SPLINE
SPL {X  -165.650, Y  +561.960, Z    +0.000, E1   +45.285, E3 +336665.881}
SPL {X  -165.650, Y  +554.065, Z    +0.000, E1   +45.254, E3 +336681.943}
SPL {X  -165.650, Y  +548.074, Z    +0.000, E1   +45.245, E3 +336694.053}
SPL {X  -165.650, Y  +542.958, Z    +0.000, E1   +45.131, E3 +336705.184}
SPL {X  -165.650, Y  +535.288, Z    +0.000, E1   +45.332, E3 +336719.625}
SPL {X  -165.650, Y  +529.160, Z    +0.000, E1   +45.215, E3 +336732.606}
SPL {X  -165.650, Y  +522.672, Z    +0.000, E1   +45.331, E3 +336745.172}
SPL {X  -165.650, Y  +516.211, Z    +0.000, E1   +45.175, E3 +336759.131}
SPL {X  -165.650, Y  +509.762, Z    +0.000, E1   +45.191, E3 +336772.174}
SPL {X  -165.650, Y  +503.812, Z    +0.000, E1   +45.188, E3 +336784.212}
SPL {X  -165.650, Y  +499.646, Z    +0.000, E1   +44.886, E3 +336794.483}
ENDSPLINE

SPLINE
SPL {X  -165.650, Y  +516.930, Z    +0.000, E1   +36.544, E3 +336803.154}
ENDSPLINE

SPLINE
SPL {X  -165.650, Y  +511.324, Z    +0.000, E1   +37.254, E3 +336814.145}
SPL {X  -165.650, Y  +504.742, Z    +0.000, E1   +38.087, E3 +336826.450}
SPL {X  -165.650, Y  +497.845, Z    +0.000, E1   +39.022, E3 +336838.525}
SPL {X  -165.650, Y  +488.971, Z    +0.000, E1   +40.149, E3 +336853.745}
SPL {X  -165.650, Y  +478.382, Z    +0.000, E1   +41.628, E3 +336869.943}
SPL {X  -165.650, Y  +472.112, Z    +0.000, E1   +42.202, E3 +336880.682}
SPL {X  -165.650, Y  +466.741, Z    +0.000, E1   +42.890, E3 +336888.603}
SPL {X  -165.650, Y  +458.202, Z    +0.000, E1   +44.020, E3 +336900.390}
SPL {X  -165.650, Y  +449.099, Z    +0.000, E1   +44.871, E3 +336914.353}
SPL {X  -165.650, Y  +442.120, Z    +0.000, E1   +45.313, E3 +336925.905}
SPL {X  -165.650, Y  +436.063, Z    +0.000, E1   +44.972, E3 +336940.489}
SPL {X  -165.650, Y  +427.943, Z    +0.000, E1   +45.362, E3 +336954.526}
SPL {X  -165.650, Y  +422.523, Z    +0.000, E1   +45.103, E3 +336967.205}
SPL {X  -165.650, Y  +415.564, Z    +0.000, E1   +45.195, E3 +336980.744}
SPL {X  -165.650, Y  +410.687, Z    +0.000, E1   +44.955, E3 +336992.060}
SPL {X  -165.650, Y  +405.522, Z    +0.000, E1   +45.119, E3 +337001.620}
SPL {X  -165.650, Y  +399.216, Z    +0.000, E1   +45.246, E3 +337013.814}
SPL {X  -165.650, Y  +391.618, Z    +0.000, E1   +45.037, E3 +337030.592}
SPL {X  -165.650, Y  +383.700, Z    +0.000, E1   +45.345, E3 +337044.718}
SPL {X  -165.650, Y  +379.225, Z    +0.000, E1   +45.073, E3 +337055.407}
SPL {X  -165.591, Y  +374.097, Z    +0.000, E1   +45.069, E3 +337065.888}
SPL {X  -165.372, Y  +368.914, Z    +0.000, E1   +45.103, E3 +337076.248}
SPL {X  -164.987, Y  +363.696, Z    +0.000, E1   +45.006, E3 +337087.471}
SPL {X  -164.256, Y  +357.053, Z    +0.000, E1   +44.969, E3 +337101.274}
SPL {X  -163.441, Y  +351.538, Z    +0.000, E1   +44.749, E3 +337113.638}
SPL {X  -162.419, Y  +345.942, Z    +0.000, E1   +44.540, E3 +337126.369}
SPL {X  -161.210, Y  +340.404, Z    +0.000, E1   +44.250, E3 +337139.194}
SPL {X  -159.961, Y  +335.460, Z    +0.000, E1   +44.205, E3 +337149.557}
SPL {X  -158.595, Y  +330.672, Z    +0.000, E1   +43.797, E3 +337161.535}
SPL {X  -157.207, Y  +326.289, Z    +0.000, E1   +43.631, E3 +337171.288}
SPL {X  -152.192, Y  +313.097, Z    +0.000, E1   +47.715, E3 +337174.842}
SPL {X  -146.385, Y  +300.967, Z    +0.000, E1   +50.402, E3 +337181.037}
SPL {X  -138.435, Y  +287.529, Z    +0.000, E1   +45.834, E3 +337242.993}
SPL {X  -134.645, Y  +282.008, Z    +0.000, E1   +45.207, E3 +337272.650}
ENDSPLINE

SPLINE
SPL {X  -154.915, Y  +319.839, Z    +0.000, E1   +31.584, E3 +337332.169}
SPL {X  -161.387, Y  +341.161, Z    +0.000, E1   +22.590, E3 +337346.014}
SPL {X  -164.566, Y  +359.576, Z    +0.000, E1   +13.425, E3 +337324.608}
SPL {X  -165.355, Y  +368.611, Z    +0.000, E1    +8.407, E3 +337328.189}
SPL {X  -165.614, Y  +375.050, Z    +0.000, E1    +4.520, E3 +337329.492}
SPL {X  -165.650, Y  +379.847, Z    +0.000, E1    +1.364, E3 +337327.842}
SPL {X  -165.650, Y  +383.246, Z    +0.000, E1    -1.216, E3 +337326.935}
SPL {X  -165.650, Y  +386.866, Z    +0.000, E1    -4.337, E3 +337326.988}
SPL {X  -165.650, Y  +394.200, Z    +0.000, E1   -11.943, E3 +337324.755}
SPL {X  -165.650, Y  +405.401, Z    +0.000, E1   -24.512, E3 +337324.575}
SPL {X  -165.650, Y  +418.038, Z    +0.000, E1   -38.688, E3 +337320.802}
SPL {X  -165.650, Y  +461.620, Z    +0.000, E1   -55.594, E3 +337340.981}
SPL {X  -165.650, Y  +498.574, Z    +0.000, E1   -52.082, E3 +337402.006}
ENDSPLINE

SPLINE
SPL {X  -165.650, Y  +484.983, Z    +0.000, E1   -45.406, E3 +337417.509}
ENDSPLINE

SPLINE
SPL {X  -165.650, Y  +492.090, Z    +0.000, E1   -45.292, E3 +337432.532}
SPL {X  -165.650, Y  +498.857, Z    +0.000, E1   -45.339, E3 +337445.869}
SPL {X  -165.650, Y  +505.115, Z    +0.000, E1   -45.299, E3 +337458.817}
SPL {X  -165.650, Y  +510.931, Z    +0.000, E1   -45.250, E3 +337470.808}
SPL {X  -165.650, Y  +516.157, Z    +0.000, E1   -45.240, E3 +337481.482}
SPL {X  -165.650, Y  +521.049, Z    +0.000, E1   -45.236, E3 +337491.435}
SPL {X  -165.650, Y  +527.050, Z    +0.000, E1   -45.345, E3 +337502.931}
SPL {X  -165.650, Y  +532.042, Z    +0.000, E1   -45.233, E3 +337513.674}
SPL {X  -165.650, Y  +537.290, Z    +0.000, E1   -45.204, E3 +337524.515}
SPL {X  -165.650, Y  +544.196, Z    +0.000, E1   -45.432, E3 +337537.189}
SPL {X  -165.650, Y  +548.678, Z    +0.000, E1   -45.162, E3 +337547.753}
SPL {X  -165.650, Y  +554.600, Z    +0.000, E1   -45.345, E3 +337558.730}
SPL {X  -165.650, Y  +559.896, Z    +0.000, E1   -45.150, E3 +337570.585}
SPL {X  -165.650, Y  +566.830, Z    +0.000, E1   -45.346, E3 +337583.566}
SPL {X  -165.650, Y  +573.074, Z    +0.000, E1   -45.379, E3 +337595.896}
SPL {X  -165.650, Y  +579.360, Z    +0.000, E1   -45.300, E3 +337609.181}
SPL {X  -165.650, Y  +584.577, Z    +0.000, E1   -45.167, E3 +337620.405}
SPL {X  -165.650, Y  +590.060, Z    +0.000, E1   -45.221, E3 +337631.295}
SPL {X  -165.650, Y  +596.611, Z    +0.000, E1   -45.390, E3 +337643.532}
SPL {X  -165.650, Y  +601.960, Z    +0.000, E1   -45.255, E3 +337655.140}
SPL {X  -165.650, Y  +605.976, Z    +0.000, E1   -45.260, E3 +337663.190}
SPL {X  -165.650, Y  +610.850, Z    +0.000, E1   -45.208, E3 +337673.459}
SPL {X  -165.650, Y  +617.450, Z    +0.000, E1   -45.402, E3 +337685.661}
SPL {X  -165.650, Y  +622.720, Z    +0.000, E1   -45.272, E3 +337697.059}
SPL {X  -165.650, Y  +627.828, Z    +0.000, E1   -45.174, E3 +337708.015}
SPL {X  -165.650, Y  +634.620, Z    +0.000, E1   -45.438, E3 +337720.221}
SPL {X  -165.650, Y  +640.808, Z    +0.000, E1   -45.294, E3 +337733.596}
SPL {X  -165.650, Y  +646.552, Z    +0.000, E1   -45.137, E3 +337746.120}
SPL {X  -165.650, Y  +652.431, Z    +0.000, E1   -45.333, E3 +337756.874}
SPL {X  -165.650, Y  +657.443, Z    +0.000, E1   -45.316, E3 +337767.131}
SPL {X  -165.650, Y  +662.999, Z    +0.000, E1   -45.214, E3 +337779.003}
SPL {X  -165.650, Y  +668.737, Z    +0.000, E1   -45.236, E3 +337790.518}
SPL {X  -165.650, Y  +675.226, Z    +0.000, E1   -45.503, E3 +337802.021}
SPL {X  -165.597, Y  +679.672, Z    +0.000, E1   -45.206, E3 +337812.742}
SPL {X  -165.388, Y  +684.808, Z    +0.000, E1   -45.192, E3 +337823.250}
SPL {X  -165.020, Y  +689.938, Z    +0.000, E1   -45.107, E3 +337834.193}
SPL {X  -164.358, Y  +696.147, Z    +0.000, E1   -45.160, E3 +337846.458}
SPL {X  -163.631, Y  +701.286, Z    +0.000, E1   -44.994, E3 +337857.751}
SPL {X  -163.047, Y  +704.748, Z    +0.000, E1   -44.682, E3 +337866.574}
SPL {X  -161.884, Y  +710.619, Z    +0.000, E1   -44.738, E3 +337878.199}
SPL {X  -160.692, Y  +715.726, Z    +0.000, E1   -44.379, E3 +337890.522}
SPL {X  -159.384, Y  +720.631, Z    +0.000, E1   -44.155, E3 +337901.672}
SPL {X  -157.745, Y  +726.062, Z    +0.000, E1   -43.902, E3 +337914.158}
SPL {X  -153.030, Y  +738.918, Z    +0.000, E1   -47.123, E3 +337921.761}
SPL {X  -145.149, Y  +755.323, Z    +0.000, E1   -51.167, E3 +337927.893}
SPL {X  -144.116, Y  +757.172, Z    +0.000, E1   -42.809, E3 +337994.443}
SPL {X  -127.227, Y  +781.582, Z    +0.000, E1   -46.780, E3 +338040.112}
ENDSPLINE

SPLINE
SPL {X  -133.736, Y  +773.248, Z    +0.000, E1   -45.385, E3 +338118.155}
SPL {X  -160.761, Y  +715.447, Z    +0.000, E1   -23.748, E3 +338075.004}
SPL {X  -164.304, Y  +696.571, Z    +0.000, E1   -14.525, E3 +338080.228}
SPL {X  -165.498, Y  +682.585, Z    +0.000, E1    -6.769, E3 +338079.903}
SPL {X  -165.650, Y  +674.975, Z    +0.000, E1    -1.888, E3 +338078.261}
SPL {X  -165.650, Y  +670.481, Z    +0.000, E1    +1.454, E3 +338077.702}
SPL {X  -165.650, Y  +665.304, Z    +0.000, E1    +6.303, E3 +338076.205}
SPL {X  -165.650, Y  +657.587, Z    +0.000, E1   +14.733, E3 +338074.979}
SPL {X  -165.650, Y  +646.511, Z    +0.000, E1   +26.434, E3 +338077.540}
SPL {X  -165.650, Y  +637.905, Z    +0.000, E1   +40.225, E3 +338065.665}
SPL {X  -165.650, Y  +607.385, Z    +0.000, E1   +51.775, E3 +338085.423}
SPL {X  -165.650, Y  +598.058, Z    +0.000, E1   +51.157, E3 +338098.884}
SPL {X  -165.650, Y  +553.219, Z    +0.000, E1   +52.865, E3 +338153.067}
ENDSPLINE

SPLINE
SPL {X  -165.650, Y  +569.883, Z    +0.000, E1   +45.183, E3 +338168.744}
ENDSPLINE

SPLINE
SPL {X  -165.650, Y  +564.081, Z    +0.000, E1   +45.208, E3 +338180.361}
SPL {X  -165.650, Y  +557.350, Z    +0.000, E1   +45.265, E3 +338193.798}
SPL {X  -165.650, Y  +549.414, Z    +0.000, E1   +45.294, E3 +338209.700}
SPL {X  -165.650, Y  +542.958, Z    +0.000, E1   +45.131, E3 +338223.702}
SPL {X  -165.650, Y  +535.288, Z    +0.000, E1   +45.332, E3 +338238.143}
SPL {X  -165.650, Y  +528.026, Z    +0.000, E1   +45.173, E3 +338253.802}
SPL {X  -165.650, Y  +519.896, Z    +0.000, E1   +45.366, E3 +338269.141}
SPL {X  -165.650, Y  +512.740, Z    +0.000, E1   +45.225, E3 +338284.488}
SPL {X  -165.650, Y  +505.100, Z    +0.000, E1   +45.197, E3 +338300.171}
SPL {X  -165.650, Y  +499.646, Z    +0.000, E1   +44.886, E3 +338313.002}
ENDSPLINE

SPLINE
SPL {X  -165.650, Y  +516.930, Z    +0.000, E1   +36.544, E3 +338321.672}
ENDSPLINE

SPLINE
SPL {X  -165.650, Y  +511.324, Z    +0.000, E1   +37.254, E3 +338332.663}
SPL {X  -165.650, Y  +502.734, Z    +0.000, E1   +38.389, E3 +338348.432}
SPL {X  -165.650, Y  +493.826, Z    +0.000, E1   +39.521, E3 +338364.094}
SPL {X  -165.650, Y  +485.086, Z    +0.000, E1   +40.678, E3 +338378.407}
SPL {X  -165.650, Y  +474.980, Z    +0.000, E1   +42.004, E3 +338394.034}
SPL {X  -165.650, Y  +463.933, Z    +0.000, E1   +43.299, E3 +338410.920}
SPL {X  -165.650, Y  +452.327, Z    +0.000, E1   +44.758, E3 +338426.826}
SPL {X  -165.650, Y  +444.380, Z    +0.000, E1   +45.056, E3 +338441.421}
SPL {X  -165.650, Y  +436.063, Z    +0.000, E1   +44.972, E3 +338459.008}
SPL {X  -165.650, Y  +427.943, Z    +0.000, E1   +45.362, E3 +338473.045}
SPL {X  -165.650, Y  +422.523, Z    +0.000, E1   +45.103, E3 +338485.723}
SPL {X  -165.650, Y  +415.564, Z    +0.000, E1   +45.195, E3 +338499.262}
SPL {X  -165.650, Y  +410.687, Z    +0.000, E1   +44.955, E3 +338510.578}
SPL {X  -165.650, Y  +405.522, Z    +0.000, E1   +45.119, E3 +338520.138}
SPL {X  -165.650, Y  +399.216, Z    +0.000, E1   +45.246, E3 +338532.332}
SPL {X  -165.650, Y  +391.618, Z    +0.000, E1   +45.037, E3 +338549.110}
SPL {X  -165.650, Y  +383.700, Z    +0.000, E1   +45.345, E3 +338563.237}
SPL {X  -165.650, Y  +379.225, Z    +0.000, E1   +45.073, E3 +338573.926}
SPL {X  -165.591, Y  +374.097, Z    +0.000, E1   +45.069, E3 +338584.407}
SPL {X  -165.372, Y  +368.914, Z    +0.000, E1   +45.103, E3 +338594.767}
SPL {X  -164.833, Y  +362.064, Z    +0.000, E1   +44.999, E3 +338609.552}
SPL {X  -164.024, Y  +355.348, Z    +0.000, E1   +45.002, E3 +338622.940}
SPL {X  -163.140, Y  +349.774, Z    +0.000, E1   +44.687, E3 +338636.327}
SPL {X  -162.065, Y  +344.224, Z    +0.000, E1   +44.509, E3 +338648.417}
SPL {X  -161.210, Y  +340.404, Z    +0.000, E1   +44.250, E3 +338657.713}
SPL {X  -159.961, Y  +335.460, Z    +0.000, E1   +44.205, E3 +338668.076}
SPL {X  -158.595, Y  +330.672, Z    +0.000, E1   +43.797, E3 +338680.054}
SPL {X  -157.207, Y  +326.289, Z    +0.000, E1   +43.631, E3 +338689.807}
SPL {X  -152.192, Y  +313.097, Z    +0.000, E1   +47.715, E3 +338693.361}
SPL {X  -146.385, Y  +300.967, Z    +0.000, E1   +50.402, E3 +338699.556}
SPL {X  -138.435, Y  +287.529, Z    +0.000, E1   +45.834, E3 +338761.512}
SPL {X  -134.645, Y  +282.008, Z    +0.000, E1   +45.207, E3 +338791.168}
ENDSPLINE

SPLINE
SPL {X  -154.915, Y  +319.839, Z    +0.000, E1   +31.584, E3 +338850.687}
SPL {X  -161.387, Y  +341.161, Z    +0.000, E1   +22.590, E3 +338864.533}
SPL {X  -164.566, Y  +359.576, Z    +0.000, E1   +13.425, E3 +338843.126}
SPL {X  -165.355, Y  +368.611, Z    +0.000, E1    +8.407, E3 +338846.707}
SPL {X  -165.614, Y  +375.050, Z    +0.000, E1    +4.520, E3 +338848.011}
SPL {X  -165.650, Y  +379.271, Z    +0.000, E1    +1.752, E3 +338845.032}
SPL {X  -165.650, Y  +382.603, Z    +0.000, E1    -0.657, E3 +338846.240}
SPL {X  -165.650, Y  +386.866, Z    +0.000, E1    -4.337, E3 +338845.506}
SPL {X  -165.650, Y  +392.464, Z    +0.000, E1   -10.170, E3 +338843.510}
SPL {X  -165.650, Y  +397.361, Z    +0.000, E1   -15.736, E3 +338842.842}
SPL {X  -165.650, Y  +404.553, Z    +0.000, E1   -23.488, E3 +338843.618}
SPL {X  -165.650, Y  +415.773, Z    +0.000, E1   -36.308, E3 +338839.770}
SPL {X  -165.650, Y  +461.620, Z    +0.000, E1   -55.594, E3 +338859.499}
SPL {X  -165.650, Y  +505.847, Z    +0.000, E1   -55.467, E3 +338911.472}
ENDSPLINE

SPLINE
SPL {X  -165.650, Y  +495.538, Z    +0.000, E1   -50.621, E3 +338923.956}
SPL {X  -165.650, Y  +483.168, Z    +0.000, E1   -45.573, E3 +338931.182}
ENDSPLINE

SPLINE
SPL {X  -165.650, Y  +487.615, Z    +0.000, E1   -45.254, E3 +338942.203}
SPL {X  -165.650, Y  +493.602, Z    +0.000, E1   -45.283, E3 +338954.043}
SPL {X  -165.650, Y  +498.857, Z    +0.000, E1   -45.339, E3 +338964.387}
SPL {X  -165.650, Y  +504.159, Z    +0.000, E1   -45.384, E3 +338974.782}
SPL {X  -165.650, Y  +509.628, Z    +0.000, E1   -45.217, E3 +338986.965}
SPL {X  -165.650, Y  +516.157, Z    +0.000, E1   -45.240, E3 +339000.000}
SPL {X  -165.650, Y  +521.049, Z    +0.000, E1   -45.236, E3 +339009.953}
SPL {X  -165.650, Y  +527.050, Z    +0.000, E1   -45.345, E3 +339021.449}
SPL {X  -165.650, Y  +532.042, Z    +0.000, E1   -45.233, E3 +339032.193}
SPL {X  -165.650, Y  +537.290, Z    +0.000, E1   -45.204, E3 +339043.033}
SPL {X  -165.650, Y  +544.196, Z    +0.000, E1   -45.432, E3 +339055.708}
SPL {X  -165.650, Y  +548.678, Z    +0.000, E1   -45.162, E3 +339066.271}
SPL {X  -165.650, Y  +554.600, Z    +0.000, E1   -45.345, E3 +339077.249}
SPL {X  -165.650, Y  +559.896, Z    +0.000, E1   -45.150, E3 +339089.104}
SPL {X  -165.650, Y  +566.830, Z    +0.000, E1   -45.346, E3 +339102.084}
SPL {X  -165.650, Y  +573.074, Z    +0.000, E1   -45.379, E3 +339114.415}
SPL {X  -165.650, Y  +577.292, Z    +0.000, E1   -45.246, E3 +339123.678}
SPL {X  -165.650, Y  +583.131, Z    +0.000, E1   -45.255, E3 +339135.620}
SPL {X  -165.650, Y  +590.060, Z    +0.000, E1   -45.221, E3 +339149.814}
SPL {X  -165.650, Y  +596.611, Z    +0.000, E1   -45.390, E3 +339162.050}
SPL {X  -165.650, Y  +603.637, Z    +0.000, E1   -45.296, E3 +339176.969}
SPL {X  -165.650, Y  +610.850, Z    +0.000, E1   -45.208, E3 +339191.977}
SPL {X  -165.650, Y  +617.450, Z    +0.000, E1   -45.402, E3 +339204.180}
SPL {X  -165.650, Y  +622.720, Z    +0.000, E1   -45.272, E3 +339215.577}
SPL {X  -165.650, Y  +627.828, Z    +0.000, E1   -45.174, E3 +339226.534}
SPL {X  -165.650, Y  +636.061, Z    +0.000, E1   -45.380, E3 +339242.196}
SPL {X  -165.650, Y  +645.149, Z    +0.000, E1   -45.285, E3 +339261.127}
SPL {X  -165.650, Y  +652.431, Z    +0.000, E1   -45.333, E3 +339275.393}
SPL {X  -165.650, Y  +657.443, Z    +0.000, E1   -45.316, E3 +339285.649}
SPL {X  -165.650, Y  +662.999, Z    +0.000, E1   -45.214, E3 +339297.521}
SPL {X  -165.650, Y  +668.737, Z    +0.000, E1   -45.236, E3 +339309.036}
SPL {X  -165.650, Y  +675.226, Z    +0.000, E1   -45.503, E3 +339320.540}
SPL {X  -165.597, Y  +679.672, Z    +0.000, E1   -45.206, E3 +339331.261}
SPL {X  -165.388, Y  +684.808, Z    +0.000, E1   -45.192, E3 +339341.768}
SPL {X  -165.020, Y  +689.938, Z    +0.000, E1   -45.107, E3 +339352.711}
SPL {X  -164.358, Y  +696.147, Z    +0.000, E1   -45.160, E3 +339364.977}
SPL {X  -163.631, Y  +701.286, Z    +0.000, E1   -44.994, E3 +339376.269}
SPL {X  -163.047, Y  +704.748, Z    +0.000, E1   -44.682, E3 +339385.093}
SPL {X  -161.884, Y  +710.619, Z    +0.000, E1   -44.738, E3 +339396.718}
SPL {X  -160.692, Y  +715.726, Z    +0.000, E1   -44.379, E3 +339409.040}
SPL {X  -158.938, Y  +722.175, Z    +0.000, E1   -44.121, E3 +339423.688}
SPL {X  -156.604, Y  +729.490, Z    +0.000, E1   -44.229, E3 +339437.678}
SPL {X  -147.100, Y  +751.668, Z    +0.000, E1   -50.624, E3 +339443.565}
SPL {X  -143.038, Y  +759.047, Z    +0.000, E1   -43.157, E3 +339515.585}
SPL {X  -123.277, Y  +786.146, Z    +0.000, E1   -47.533, E3 +339571.640}
ENDSPLINE

SPLINE
SPL {X  -133.736, Y  +773.248, Z    +0.000, E1   -45.385, E3 +339636.673}
SPL {X  -160.761, Y  +715.447, Z    +0.000, E1   -23.748, E3 +339593.523}
SPL {X  -164.304, Y  +696.571, Z    +0.000, E1   -14.525, E3 +339598.747}
SPL {X  -165.374, Y  +685.052, Z    +0.000, E1    -8.166, E3 +339598.140}
SPL {X  -165.648, Y  +676.230, Z    +0.000, E1    -2.814, E3 +339597.292}
SPL {X  -165.650, Y  +670.481, Z    +0.000, E1    +1.454, E3 +339596.221}
SPL {X  -165.650, Y  +665.304, Z    +0.000, E1    +6.303, E3 +339594.723}
SPL {X  -165.650, Y  +657.587, Z    +0.000, E1   +14.733, E3 +339593.498}
SPL {X  -165.650, Y  +646.511, Z    +0.000, E1   +26.434, E3 +339596.059}
SPL {X  -165.650, Y  +637.905, Z    +0.000, E1   +40.225, E3 +339584.183}
SPL {X  -165.650, Y  +607.385, Z    +0.000, E1   +51.775, E3 +339603.941}
SPL {X  -165.650, Y  +598.058, Z    +0.000, E1   +51.157, E3 +339617.403}
SPL {X  -165.650, Y  +553.656, Z    +0.000, E1   +53.998, E3 +339664.402}
SPL {X  -165.650, Y  +553.154, Z    +0.000, E1   +52.102, E3 +339675.929}
ENDSPLINE

SPLINE
SPL {X  -165.650, Y  +569.883, Z    +0.000, E1   +45.183, E3 +339687.262}
ENDSPLINE

SPLINE
SPL {X  -165.650, Y  +564.081, Z    +0.000, E1   +45.208, E3 +339698.880}
SPL {X  -165.650, Y  +557.350, Z    +0.000, E1   +45.265, E3 +339712.317}
SPL {X  -165.650, Y  +549.414, Z    +0.000, E1   +45.294, E3 +339728.219}
SPL {X  -165.650, Y  +542.958, Z    +0.000, E1   +45.131, E3 +339742.221}
SPL {X  -165.650, Y  +535.288, Z    +0.000, E1   +45.332, E3 +339756.662}
SPL {X  -165.650, Y  +528.026, Z    +0.000, E1   +45.173, E3 +339772.320}
SPL {X  -165.650, Y  +520.964, Z    +0.000, E1   +45.458, E3 +339784.825}
SPL {X  -165.650, Y  +516.211, Z    +0.000, E1   +45.175, E3 +339796.168}
SPL {X  -165.650, Y  +509.762, Z    +0.000, E1   +45.191, E3 +339809.211}
SPL {X  -165.650, Y  +503.812, Z    +0.000, E1   +45.188, E3 +339821.249}
SPL {X  -165.650, Y  +499.646, Z    +0.000, E1   +44.886, E3 +339831.520}
ENDSPLINE

SPLINE
SPL {X  -165.650, Y  +516.930, Z    +0.000, E1   +36.544, E3 +339840.191}
ENDSPLINE

SPLINE
SPL {X  -165.650, Y  +511.324, Z    +0.000, E1   +37.254, E3 +339851.182}
SPL {X  -165.650, Y  +504.742, Z    +0.000, E1   +38.087, E3 +339863.487}
SPL {X  -165.650, Y  +497.845, Z    +0.000, E1   +39.022, E3 +339875.562}
SPL {X  -165.650, Y  +488.971, Z    +0.000, E1   +40.149, E3 +339890.783}
SPL {X  -165.650, Y  +478.382, Z    +0.000, E1   +41.628, E3 +339906.980}
SPL {X  -165.650, Y  +472.112, Z    +0.000, E1   +42.202, E3 +339917.719}
SPL {X  -165.650, Y  +466.741, Z    +0.000, E1   +42.890, E3 +339925.640}
SPL {X  -165.650, Y  +458.202, Z    +0.000, E1   +44.020, E3 +339937.427}
SPL {X  -165.650, Y  +449.099, Z    +0.000, E1   +44.871, E3 +339951.390}
SPL {X  -165.650, Y  +442.120, Z    +0.000, E1   +45.313, E3 +339962.942}
SPL {X  -165.650, Y  +436.063, Z    +0.000, E1   +44.972, E3 +339977.526}
SPL {X  -165.650, Y  +427.943, Z    +0.000, E1   +45.362, E3 +339991.563}
SPL {X  -165.650, Y  +422.523, Z    +0.000, E1   +45.103, E3 +340004.242}
SPL {X  -165.650, Y  +415.564, Z    +0.000, E1   +45.195, E3 +340017.781}
SPL {X  -165.650, Y  +410.687, Z    +0.000, E1   +44.955, E3 +340029.097}
SPL {X  -165.650, Y  +405.522, Z    +0.000, E1   +45.119, E3 +340038.657}
SPL {X  -165.650, Y  +400.300, Z    +0.000, E1   +45.439, E3 +340047.341}
SPL {X  -165.650, Y  +396.171, Z    +0.000, E1   +44.969, E3 +340058.598}
SPL {X  -165.650, Y  +390.060, Z    +0.000, E1   +45.007, E3 +340070.832}
SPL {X  -165.650, Y  +383.700, Z    +0.000, E1   +45.345, E3 +340081.755}
SPL {X  -165.650, Y  +379.225, Z    +0.000, E1   +45.073, E3 +340092.444}
SPL {X  -165.591, Y  +374.097, Z    +0.000, E1   +45.069, E3 +340102.926}
SPL {X  -165.372, Y  +368.914, Z    +0.000, E1   +45.103, E3 +340113.285}
SPL {X  -164.833, Y  +362.064, Z    +0.000, E1   +44.999, E3 +340128.070}
SPL {X  -164.024, Y  +355.348, Z    +0.000, E1   +45.002, E3 +340141.459}
SPL {X  -163.441, Y  +351.538, Z    +0.000, E1   +44.749, E3 +340150.675}
SPL {X  -162.419, Y  +345.942, Z    +0.000, E1   +44.540, E3 +340163.406}
SPL {X  -161.210, Y  +340.404, Z    +0.000, E1   +44.250, E3 +340176.231}
SPL {X  -159.961, Y  +335.460, Z    +0.000, E1   +44.205, E3 +340186.594}
SPL {X  -158.595, Y  +330.672, Z    +0.000, E1   +43.797, E3 +340198.572}
SPL {X  -156.695, Y  +324.773, Z    +0.000, E1   +43.987, E3 +340209.469}
SPL {X  -148.318, Y  +304.733, Z    +0.000, E1   +49.897, E3 +340214.706}
SPL {X  -137.641, Y  +286.333, Z    +0.000, E1   +45.396, E3 +340289.566}
SPL {X  -137.518, Y  +286.149, Z    +0.000, E1   +42.648, E3 +340362.075}
ENDSPLINE

SPLINE
SPL {X  -156.430, Y  +324.005, Z    +0.000, E1   +29.926, E3 +340367.210}
SPL {X  -161.387, Y  +341.161, Z    +0.000, E1   +22.590, E3 +340383.051}
SPL {X  -164.566, Y  +359.576, Z    +0.000, E1   +13.425, E3 +340361.645}
SPL {X  -165.355, Y  +368.611, Z    +0.000, E1    +8.407, E3 +340365.226}
SPL {X  -165.614, Y  +375.050, Z    +0.000, E1    +4.520, E3 +340366.529}
SPL {X  -165.650, Y  +379.271, Z    +0.000, E1    +1.752, E3 +340363.551}
SPL {X  -165.650, Y  +382.603, Z    +0.000, E1    -0.657, E3 +340364.759}
SPL {X  -165.650, Y  +386.866, Z    +0.000, E1    -4.337, E3 +340364.025}
SPL {X  -165.650, Y  +394.200, Z    +0.000, E1   -11.943, E3 +340361.792}
SPL {X  -165.650, Y  +405.401, Z    +0.000, E1   -24.512, E3 +340361.612}
SPL {X  -165.650, Y  +418.038, Z    +0.000, E1   -38.688, E3 +340357.839}
SPL {X  -165.650, Y  +461.620, Z    +0.000, E1   -55.594, E3 +340378.018}
SPL {X  -165.650, Y  +498.574, Z    +0.000, E1   -52.082, E3 +340439.043}
ENDSPLINE

SPLINE
SPL {X  -165.650, Y  +483.168, Z    +0.000, E1   -45.573, E3 +340449.700}
ENDSPLINE

SPLINE
SPL {X  -165.650, Y  +487.615, Z    +0.000, E1   -45.254, E3 +340460.722}
SPL {X  -165.650, Y  +493.602, Z    +0.000, E1   -45.283, E3 +340472.562}
SPL {X  -165.650, Y  +498.857, Z    +0.000, E1   -45.339, E3 +340482.906}
SPL {X  -165.650, Y  +504.159, Z    +0.000, E1   -45.384, E3 +340493.300}
SPL {X  -165.650, Y  +509.628, Z    +0.000, E1   -45.217, E3 +340505.483}
SPL {X  -165.650, Y  +516.157, Z    +0.000, E1   -45.240, E3 +340518.519}
SPL {X  -165.650, Y  +521.049, Z    +0.000, E1   -45.236, E3 +340528.472}
SPL {X  -165.650, Y  +527.050, Z    +0.000, E1   -45.345, E3 +340539.968}
SPL {X  -165.650, Y  +532.042, Z    +0.000, E1   -45.233, E3 +340550.711}
SPL {X  -165.650, Y  +537.290, Z    +0.000, E1   -45.204, E3 +340561.552}
SPL {X  -165.650, Y  +544.196, Z    +0.000, E1   -45.432, E3 +340574.226}
SPL {X  -165.650, Y  +548.678, Z    +0.000, E1   -45.162, E3 +340584.790}
SPL {X  -165.650, Y  +554.600, Z    +0.000, E1   -45.345, E3 +340595.767}
SPL {X  -165.650, Y  +559.896, Z    +0.000, E1   -45.150, E3 +340607.622}
SPL {X  -165.650, Y  +566.830, Z    +0.000, E1   -45.346, E3 +340620.603}
SPL {X  -165.650, Y  +573.074, Z    +0.000, E1   -45.379, E3 +340632.933}
SPL {X  -165.650, Y  +579.360, Z    +0.000, E1   -45.300, E3 +340646.218}
SPL {X  -165.650, Y  +584.577, Z    +0.000, E1   -45.167, E3 +340657.442}
SPL {X  -165.650, Y  +590.060, Z    +0.000, E1   -45.221, E3 +340668.333}
SPL {X  -165.650, Y  +596.611, Z    +0.000, E1   -45.390, E3 +340680.569}
SPL {X  -165.650, Y  +601.960, Z    +0.000, E1   -45.255, E3 +340692.177}
SPL {X  -165.650, Y  +605.976, Z    +0.000, E1   -45.260, E3 +340700.227}
SPL {X  -165.650, Y  +610.850, Z    +0.000, E1   -45.208, E3 +340710.496}
SPL {X  -165.650, Y  +617.450, Z    +0.000, E1   -45.402, E3 +340722.698}
SPL {X  -165.650, Y  +622.720, Z    +0.000, E1   -45.272, E3 +340734.096}
SPL {X  -165.650, Y  +627.828, Z    +0.000, E1   -45.174, E3 +340745.053}
SPL {X  -165.650, Y  +634.620, Z    +0.000, E1   -45.438, E3 +340757.258}
SPL {X  -165.650, Y  +640.808, Z    +0.000, E1   -45.294, E3 +340770.633}
SPL {X  -165.650, Y  +646.552, Z    +0.000, E1   -45.137, E3 +340783.157}
SPL {X  -165.650, Y  +652.431, Z    +0.000, E1   -45.333, E3 +340793.911}
SPL {X  -165.650, Y  +657.443, Z    +0.000, E1   -45.316, E3 +340804.168}
SPL {X  -165.650, Y  +662.999, Z    +0.000, E1   -45.214, E3 +340816.040}
SPL {X  -165.650, Y  +668.737, Z    +0.000, E1   -45.236, E3 +340827.555}
SPL {X  -165.650, Y  +675.226, Z    +0.000, E1   -45.503, E3 +340839.058}
SPL {X  -165.597, Y  +679.672, Z    +0.000, E1   -45.206, E3 +340849.779}
SPL {X  -165.388, Y  +684.808, Z    +0.000, E1   -45.192, E3 +340860.287}
SPL {X  -165.020, Y  +689.938, Z    +0.000, E1   -45.107, E3 +340871.230}
SPL {X  -164.358, Y  +696.147, Z    +0.000, E1   -45.160, E3 +340883.495}
SPL {X  -163.631, Y  +701.286, Z    +0.000, E1   -44.994, E3 +340894.788}
SPL {X  -163.047, Y  +704.748, Z    +0.000, E1   -44.682, E3 +340903.611}
SPL {X  -161.884, Y  +710.619, Z    +0.000, E1   -44.738, E3 +340915.236}
SPL {X  -160.692, Y  +715.726, Z    +0.000, E1   -44.379, E3 +340927.559}
SPL {X  -159.384, Y  +720.631, Z    +0.000, E1   -44.155, E3 +340938.709}
SPL {X  -157.745, Y  +726.062, Z    +0.000, E1   -43.902, E3 +340951.195}
SPL {X  -153.030, Y  +738.918, Z    +0.000, E1   -47.123, E3 +340958.798}
SPL {X  -145.149, Y  +755.323, Z    +0.000, E1   -51.167, E3 +340964.930}
SPL {X  -143.038, Y  +759.047, Z    +0.000, E1   -43.157, E3 +341034.104}
SPL {X  -123.277, Y  +786.146, Z    +0.000, E1   -47.533, E3 +341090.159}
ENDSPLINE

SPLINE
SPL {X  -133.736, Y  +773.248, Z    +0.000, E1   -45.385, E3 +341155.192}
SPL {X  -160.761, Y  +715.447, Z    +0.000, E1   -23.748, E3 +341112.041}
SPL {X  -164.304, Y  +696.571, Z    +0.000, E1   -14.525, E3 +341117.265}
SPL {X  -165.374, Y  +685.052, Z    +0.000, E1    -8.166, E3 +341116.659}
SPL {X  -165.648, Y  +676.230, Z    +0.000, E1    -2.814, E3 +341115.810}
SPL {X  -165.650, Y  +670.481, Z    +0.000, E1    +1.454, E3 +341114.739}
SPL {X  -165.650, Y  +665.304, Z    +0.000, E1    +6.303, E3 +341113.242}
SPL {X  -165.650, Y  +657.587, Z    +0.000, E1   +14.733, E3 +341112.016}
SPL {X  -165.650, Y  +646.511, Z    +0.000, E1   +26.434, E3 +341114.577}
SPL {X  -165.650, Y  +637.905, Z    +0.000, E1   +40.225, E3 +341102.702}
SPL {X  -165.650, Y  +607.385, Z    +0.000, E1   +51.775, E3 +341122.460}
SPL {X  -165.650, Y  +598.058, Z    +0.000, E1   +51.157, E3 +341135.921}
SPL {X  -165.650, Y  +553.656, Z    +0.000, E1   +53.998, E3 +341182.921}
SPL {X  -165.650, Y  +553.154, Z    +0.000, E1   +52.102, E3 +341194.448}
ENDSPLINE

SPLINE
SPL {X  -165.650, Y  +569.883, Z    +0.000, E1   +45.183, E3 +341205.781}
ENDSPLINE

SPLINE
SPL {X  -165.650, Y  +564.081, Z    +0.000, E1   +45.208, E3 +341217.398}
SPL {X  -165.650, Y  +557.350, Z    +0.000, E1   +45.265, E3 +341230.835}
SPL {X  -165.650, Y  +549.414, Z    +0.000, E1   +45.294, E3 +341246.737}
SPL {X  -165.650, Y  +542.958, Z    +0.000, E1   +45.131, E3 +341260.740}
SPL {X  -165.650, Y  +535.288, Z    +0.000, E1   +45.332, E3 +341275.180}
SPL {X  -165.650, Y  +528.026, Z    +0.000, E1   +45.173, E3 +341290.839}
SPL {X  -165.650, Y  +520.964, Z    +0.000, E1   +45.458, E3 +341303.344}
SPL {X  -165.650, Y  +516.211, Z    +0.000, E1   +45.175, E3 +341314.687}
SPL {X  -165.650, Y  +511.047, Z    +0.000, E1   +45.193, E3 +341325.005}
SPL {X  -165.650, Y  +505.100, Z    +0.000, E1   +45.197, E3 +341337.208}
SPL {X  -165.650, Y  +499.646, Z    +0.000, E1   +44.886, E3 +341350.039}
ENDSPLINE

SPLINE
SPL {X  -165.650, Y  +516.930, Z    +0.000, E1   +36.544, E3 +341358.709}
ENDSPLINE

SPLINE
SPL {X  -165.650, Y  +511.324, Z    +0.000, E1   +37.254, E3 +341369.700}
SPL {X  -165.650, Y  +502.734, Z    +0.000, E1   +38.389, E3 +341385.469}
SPL {X  -165.650, Y  +493.826, Z    +0.000, E1   +39.521, E3 +341401.131}
SPL {X  -165.650, Y  +485.086, Z    +0.000, E1   +40.678, E3 +341415.444}
SPL {X  -165.650, Y  +476.633, Z    +0.000, E1   +41.847, E3 +341428.143}
SPL {X  -165.650, Y  +468.596, Z    +0.000, E1   +42.673, E3 +341441.405}
SPL {X  -165.650, Y  +460.562, Z    +0.000, E1   +43.733, E3 +341452.557}
SPL {X  -165.650, Y  +455.629, Z    +0.000, E1   +44.293, E3 +341459.676}
SPL {X  -165.650, Y  +449.099, Z    +0.000, E1   +44.871, E3 +341469.908}
SPL {X  -165.650, Y  +442.120, Z    +0.000, E1   +45.313, E3 +341481.460}
SPL {X  -165.650, Y  +436.063, Z    +0.000, E1   +44.972, E3 +341496.045}
SPL {X  -165.650, Y  +427.943, Z    +0.000, E1   +45.362, E3 +341510.082}
SPL {X  -165.650, Y  +422.523, Z    +0.000, E1   +45.103, E3 +341522.760}
SPL {X  -165.650, Y  +415.564, Z    +0.000, E1   +45.195, E3 +341536.299}
SPL {X  -165.650, Y  +410.687, Z    +0.000, E1   +44.955, E3 +341547.615}
SPL {X  -165.650, Y  +405.522, Z    +0.000, E1   +45.119, E3 +341557.175}
SPL {X  -165.650, Y  +399.216, Z    +0.000, E1   +45.246, E3 +341569.369}
SPL {X  -165.650, Y  +391.618, Z    +0.000, E1   +45.037, E3 +341586.147}
SPL {X  -165.650, Y  +383.700, Z    +0.000, E1   +45.345, E3 +341600.274}
SPL {X  -165.650, Y  +379.225, Z    +0.000, E1   +45.073, E3 +341610.963}
SPL {X  -165.591, Y  +374.097, Z    +0.000, E1   +45.069, E3 +341621.444}
SPL {X  -165.372, Y  +368.914, Z    +0.000, E1   +45.103, E3 +341631.804}
SPL {X  -164.987, Y  +363.696, Z    +0.000, E1   +45.006, E3 +341643.027}
SPL {X  -164.256, Y  +357.053, Z    +0.000, E1   +44.969, E3 +341656.830}
SPL {X  -163.441, Y  +351.538, Z    +0.000, E1   +44.749, E3 +341669.193}
SPL {X  -162.419, Y  +345.942, Z    +0.000, E1   +44.540, E3 +341681.925}
SPL {X  -161.210, Y  +340.404, Z    +0.000, E1   +44.250, E3 +341694.750}
SPL {X  -159.961, Y  +335.460, Z    +0.000, E1   +44.205, E3 +341705.113}
SPL {X  -158.595, Y  +330.672, Z    +0.000, E1   +43.797, E3 +341717.091}
SPL {X  -156.695, Y  +324.773, Z    +0.000, E1   +43.987, E3 +341727.988}
SPL {X  -148.318, Y  +304.733, Z    +0.000, E1   +49.897, E3 +341733.224}
SPL {X  -138.435, Y  +287.529, Z    +0.000, E1   +45.834, E3 +341798.549}
SPL {X  -134.645, Y  +282.008, Z    +0.000, E1   +45.207, E3 +341828.205}
ENDSPLINE

SPLINE
SPL {X  -154.915, Y  +319.839, Z    +0.000, E1   +31.584, E3 +341887.724}
SPL {X  -161.387, Y  +341.161, Z    +0.000, E1   +22.590, E3 +341901.570}
SPL {X  -164.566, Y  +359.576, Z    +0.000, E1   +13.425, E3 +341880.163}
SPL {X  -165.355, Y  +368.611, Z    +0.000, E1    +8.407, E3 +341883.744}
SPL {X  -165.614, Y  +375.050, Z    +0.000, E1    +4.520, E3 +341885.048}
SPL {X  -165.650, Y  +379.847, Z    +0.000, E1    +1.364, E3 +341883.397}
SPL {X  -165.650, Y  +383.246, Z    +0.000, E1    -1.216, E3 +341882.491}
SPL {X  -165.650, Y  +386.866, Z    +0.000, E1    -4.337, E3 +341882.543}
SPL {X  -165.650, Y  +394.200, Z    +0.000, E1   -11.943, E3 +341880.310}
SPL {X  -165.650, Y  +405.401, Z    +0.000, E1   -24.512, E3 +341880.130}
SPL {X  -165.650, Y  +418.038, Z    +0.000, E1   -38.688, E3 +341876.358}
SPL {X  -165.650, Y  +461.620, Z    +0.000, E1   -55.594, E3 +341896.536}
SPL {X  -165.650, Y  +505.847, Z    +0.000, E1   -55.467, E3 +341948.509}
ENDSPLINE

SPLINE
SPL {X  -165.650, Y  +495.538, Z    +0.000, E1   -50.621, E3 +341960.993}
SPL {X  -165.650, Y  +483.168, Z    +0.000, E1   -45.573, E3 +341968.219}
ENDSPLINE

SPLINE
SPL {X  -165.650, Y  +487.615, Z    +0.000, E1   -45.254, E3 +341979.240}
SPL {X  -165.650, Y  +493.602, Z    +0.000, E1   -45.283, E3 +341991.080}
SPL {X  -165.650, Y  +498.857, Z    +0.000, E1   -45.339, E3 +342001.424}
SPL {X  -165.650, Y  +504.159, Z    +0.000, E1   -45.384, E3 +342011.819}
SPL {X  -165.650, Y  +509.628, Z    +0.000, E1   -45.217, E3 +342024.002}
SPL {X  -165.650, Y  +516.157, Z    +0.000, E1   -45.240, E3 +342037.037}
SPL {X  -165.650, Y  +521.049, Z    +0.000, E1   -45.236, E3 +342046.990}
SPL {X  -165.650, Y  +527.050, Z    +0.000, E1   -45.345, E3 +342058.486}
SPL {X  -165.650, Y  +532.042, Z    +0.000, E1   -45.233, E3 +342069.230}
SPL {X  -165.650, Y  +537.290, Z    +0.000, E1   -45.204, E3 +342080.070}
SPL {X  -165.650, Y  +544.196, Z    +0.000, E1   -45.432, E3 +342092.745}
SPL {X  -165.650, Y  +548.678, Z    +0.000, E1   -45.162, E3 +342103.308}
SPL {X  -165.650, Y  +554.600, Z    +0.000, E1   -45.345, E3 +342114.286}
SPL {X  -165.650, Y  +559.896, Z    +0.000, E1   -45.150, E3 +342126.141}
SPL {X  -165.650, Y  +566.830, Z    +0.000, E1   -45.346, E3 +342139.121}
SPL {X  -165.650, Y  +573.074, Z    +0.000, E1   -45.379, E3 +342151.452}
SPL {X  -165.650, Y  +577.292, Z    +0.000, E1   -45.246, E3 +342160.715}
SPL {X  -165.650, Y  +583.131, Z    +0.000, E1   -45.255, E3 +342172.657}
SPL {X  -165.650, Y  +590.060, Z    +0.000, E1   -45.221, E3 +342186.851}
SPL {X  -165.650, Y  +596.611, Z    +0.000, E1   -45.390, E3 +342199.087}
SPL {X  -165.650, Y  +603.637, Z    +0.000, E1   -45.296, E3 +342214.006}
SPL {X  -165.650, Y  +610.850, Z    +0.000, E1   -45.208, E3 +342229.014}
SPL {X  -165.650, Y  +617.450, Z    +0.000, E1   -45.402, E3 +342241.217}
SPL {X  -165.650, Y  +622.720, Z    +0.000, E1   -45.272, E3 +342252.614}
SPL {X  -165.650, Y  +627.828, Z    +0.000, E1   -45.174, E3 +342263.571}
SPL {X  -165.650, Y  +634.620, Z    +0.000, E1   -45.438, E3 +342275.777}
SPL {X  -165.650, Y  +640.808, Z    +0.000, E1   -45.294, E3 +342289.151}
SPL {X  -165.650, Y  +646.552, Z    +0.000, E1   -45.137, E3 +342301.675}
SPL {X  -165.650, Y  +652.431, Z    +0.000, E1   -45.333, E3 +342312.430}
SPL {X  -165.650, Y  +657.443, Z    +0.000, E1   -45.316, E3 +342322.686}
SPL {X  -165.650, Y  +662.999, Z    +0.000, E1   -45.214, E3 +342334.558}
SPL {X  -165.650, Y  +668.737, Z    +0.000, E1   -45.236, E3 +342346.073}
SPL {X  -165.650, Y  +675.226, Z    +0.000, E1   -45.503, E3 +342357.577}
SPL {X  -165.597, Y  +679.672, Z    +0.000, E1   -45.206, E3 +342368.298}
SPL {X  -165.388, Y  +684.808, Z    +0.000, E1   -45.192, E3 +342378.805}
SPL {X  -165.020, Y  +689.938, Z    +0.000, E1   -45.107, E3 +342389.748}
SPL {X  -164.358, Y  +696.147, Z    +0.000, E1   -45.160, E3 +342402.014}
SPL {X  -163.631, Y  +701.286, Z    +0.000, E1   -44.994, E3 +342413.306}
SPL {X  -163.047, Y  +704.748, Z    +0.000, E1   -44.682, E3 +342422.130}
SPL {X  -161.884, Y  +710.619, Z    +0.000, E1   -44.738, E3 +342433.755}
SPL {X  -160.692, Y  +715.726, Z    +0.000, E1   -44.379, E3 +342446.077}
SPL {X  -159.384, Y  +720.631, Z    +0.000, E1   -44.155, E3 +342457.227}
SPL {X  -157.745, Y  +726.062, Z    +0.000, E1   -43.902, E3 +342469.714}
SPL {X  -153.030, Y  +738.918, Z    +0.000, E1   -47.123, E3 +342477.316}
SPL {X  -145.149, Y  +755.323, Z    +0.000, E1   -51.167, E3 +342483.448}
SPL {X  -144.116, Y  +757.172, Z    +0.000, E1   -42.809, E3 +342549.998}
SPL {X  -127.227, Y  +781.582, Z    +0.000, E1   -46.780, E3 +342595.668}
ENDSPLINE

SPLINE
SPL {X  -133.736, Y  +773.248, Z    +0.000, E1   -45.385, E3 +342673.710}
SPL {X  -160.761, Y  +715.447, Z    +0.000, E1   -23.748, E3 +342630.560}
SPL {X  -164.304, Y  +696.571, Z    +0.000, E1   -14.525, E3 +342635.784}
SPL {X  -165.374, Y  +685.052, Z    +0.000, E1    -8.166, E3 +342635.178}
SPL {X  -165.648, Y  +676.230, Z    +0.000, E1    -2.814, E3 +342634.329}
SPL {X  -165.650, Y  +670.481, Z    +0.000, E1    +1.454, E3 +342633.258}
SPL {X  -165.650, Y  +665.304, Z    +0.000, E1    +6.303, E3 +342631.760}
SPL {X  -165.650, Y  +660.688, Z    +0.000, E1   +11.392, E3 +342630.893}
SPL {X  -165.650, Y  +655.692, Z    +0.000, E1   +17.061, E3 +342630.316}
SPL {X  -165.650, Y  +646.511, Z    +0.000, E1   +26.434, E3 +342633.096}
SPL {X  -165.650, Y  +637.905, Z    +0.000, E1   +40.225, E3 +342621.220}
SPL {X  -165.650, Y  +607.385, Z    +0.000, E1   +51.775, E3 +342640.978}
SPL {X  -165.650, Y  +598.058, Z    +0.000, E1   +51.157, E3 +342654.440}
SPL {X  -165.650, Y  +553.219, Z    +0.000, E1   +52.865, E3 +342708.622}
ENDSPLINE

SPLINE
SPL {X  -165.650, Y  +569.883, Z    +0.000, E1   +45.183, E3 +342724.299}
ENDSPLINE

SPLINE
SPL {X  -165.650, Y  +564.081, Z    +0.000, E1   +45.208, E3 +342735.917}
SPL {X  -165.650, Y  +557.350, Z    +0.000, E1   +45.265, E3 +342749.354}
SPL {X  -165.650, Y  +549.414, Z    +0.000, E1   +45.294, E3 +342765.256}
SPL {X  -165.650, Y  +542.958, Z    +0.000, E1   +45.131, E3 +342779.258}
SPL {X  -165.650, Y  +535.288, Z    +0.000, E1   +45.332, E3 +342793.699}
SPL {X  -165.650, Y  +528.026, Z    +0.000, E1   +45.173, E3 +342809.357}
SPL {X  -165.650, Y  +520.964, Z    +0.000, E1   +45.458, E3 +342821.862}
SPL {X  -165.650, Y  +516.211, Z    +0.000, E1   +45.175, E3 +342833.205}
SPL {X  -165.650, Y  +511.047, Z    +0.000, E1   +45.193, E3 +342843.524}
SPL {X  -165.650, Y  +505.100, Z    +0.000, E1   +45.197, E3 +342855.727}
SPL {X  -165.650, Y  +499.646, Z    +0.000, E1   +44.886, E3 +342868.557}
ENDSPLINE

SPLINE
SPL {X  -165.650, Y  +514.834, Z    +0.000, E1   +36.829, E3 +342881.323}
ENDSPLINE

SPLINE
SPL {X  -165.650, Y  +506.421, Z    +0.000, E1   +37.886, E3 +342897.435}
SPL {X  -165.650, Y  +499.917, Z    +0.000, E1   +38.752, E3 +342908.896}
SPL {X  -165.650, Y  +493.826, Z    +0.000, E1   +39.521, E3 +342919.650}
SPL {X  -165.650, Y  +487.003, Z    +0.000, E1   +40.380, E3 +342931.104}
SPL {X  -165.650, Y  +478.382, Z    +0.000, E1   +41.628, E3 +342944.017}
SPL {X  -165.650, Y  +472.112, Z    +0.000, E1   +42.202, E3 +342954.756}
SPL {X  -165.650, Y  +466.741, Z    +0.000, E1   +42.890, E3 +342962.677}
SPL {X  -165.650, Y  +458.202, Z    +0.000, E1   +44.020, E3 +342974.465}
SPL {X  -165.650, Y  +449.099, Z    +0.000, E1   +44.871, E3 +342988.427}
SPL {X  -165.650, Y  +442.120, Z    +0.000, E1   +45.313, E3 +342999.979}
SPL {X  -165.650, Y  +436.063, Z    +0.000, E1   +44.972, E3 +343014.563}
SPL {X  -165.650, Y  +427.943, Z    +0.000, E1   +45.362, E3 +343028.600}
SPL {X  -165.650, Y  +422.523, Z    +0.000, E1   +45.103, E3 +343041.279}
SPL {X  -165.650, Y  +415.564, Z    +0.000, E1   +45.195, E3 +343054.818}
SPL {X  -165.650, Y  +410.687, Z    +0.000, E1   +44.955, E3 +343066.134}
SPL {X  -165.650, Y  +405.522, Z    +0.000, E1   +45.119, E3 +343075.694}
SPL {X  -165.650, Y  +399.216, Z    +0.000, E1   +45.246, E3 +343087.888}
SPL {X  -165.650, Y  +391.618, Z    +0.000, E1   +45.037, E3 +343104.666}
SPL {X  -165.650, Y  +383.700, Z    +0.000, E1   +45.345, E3 +343118.792}
SPL {X  -165.650, Y  +379.225, Z    +0.000, E1   +45.073, E3 +343129.482}
SPL {X  -165.591, Y  +374.097, Z    +0.000, E1   +45.069, E3 +343139.963}
SPL {X  -165.372, Y  +368.914, Z    +0.000, E1   +45.103, E3 +343150.322}
SPL {X  -164.987, Y  +363.696, Z    +0.000, E1   +45.006, E3 +343161.545}
SPL {X  -164.256, Y  +357.053, Z    +0.000, E1   +44.969, E3 +343175.348}
SPL {X  -163.441, Y  +351.538, Z    +0.000, E1   +44.749, E3 +343187.712}
SPL {X  -162.419, Y  +345.942, Z    +0.000, E1   +44.540, E3 +343200.443}
SPL {X  -161.210, Y  +340.404, Z    +0.000, E1   +44.250, E3 +343213.268}
SPL {X  -159.961, Y  +335.460, Z    +0.000, E1   +44.205, E3 +343223.631}
SPL {X  -158.595, Y  +330.672, Z    +0.000, E1   +43.797, E3 +343235.609}
SPL {X  -156.695, Y  +324.773, Z    +0.000, E1   +43.987, E3 +343246.506}
SPL {X  -148.318, Y  +304.733, Z    +0.000, E1   +49.897, E3 +343251.743}
SPL {X  -138.435, Y  +287.529, Z    +0.000, E1   +45.834, E3 +343317.067}
SPL {X  -134.645, Y  +282.008, Z    +0.000, E1   +45.207, E3 +343346.724}
ENDSPLINE

SPLINE
SPL {X  -154.915, Y  +319.839, Z    +0.000, E1   +31.584, E3 +343406.243}
SPL {X  -161.387, Y  +341.161, Z    +0.000, E1   +22.590, E3 +343420.088}
SPL {X  -164.566, Y  +359.576, Z    +0.000, E1   +13.425, E3 +343398.682}
SPL {X  -165.355, Y  +368.611, Z    +0.000, E1    +8.407, E3 +343402.263}
SPL {X  -165.614, Y  +375.050, Z    +0.000, E1    +4.520, E3 +343403.566}
SPL {X  -165.650, Y  +379.271, Z    +0.000, E1    +1.752, E3 +343400.588}
SPL {X  -165.650, Y  +382.603, Z    +0.000, E1    -0.657, E3 +343401.796}
SPL {X  -165.650, Y  +386.866, Z    +0.000, E1    -4.337, E3 +343401.062}
SPL {X  -165.650, Y  +394.200, Z    +0.000, E1   -11.943, E3 +343398.829}
SPL {X  -165.650, Y  +405.401, Z    +0.000, E1   -24.512, E3 +343398.649}
SPL {X  -165.650, Y  +418.038, Z    +0.000, E1   -38.688, E3 +343394.876}
SPL {X  -165.650, Y  +461.620, Z    +0.000, E1   -55.594, E3 +343415.055}
SPL {X  -165.650, Y  +498.574, Z    +0.000, E1   -52.082, E3 +343476.080}
ENDSPLINE

SPLINE
SPL {X  -165.650, Y  +483.168, Z    +0.000, E1   -45.573, E3 +343486.737}
ENDSPLINE

SPLINE
SPL {X  -165.650, Y  +487.615, Z    +0.000, E1   -45.254, E3 +343497.759}
SPL {X  -165.650, Y  +493.602, Z    +0.000, E1   -45.283, E3 +343509.599}
SPL {X  -165.650, Y  +498.857, Z    +0.000, E1   -45.339, E3 +343519.943}
SPL {X  -165.650, Y  +504.159, Z    +0.000, E1   -45.384, E3 +343530.337}
SPL {X  -165.650, Y  +509.628, Z    +0.000, E1   -45.217, E3 +343542.520}
SPL {X  -165.650, Y  +516.157, Z    +0.000, E1   -45.240, E3 +343555.556}
SPL {X  -165.650, Y  +521.049, Z    +0.000, E1   -45.236, E3 +343565.509}
SPL {X  -165.650, Y  +527.050, Z    +0.000, E1   -45.345, E3 +343577.005}
SPL {X  -165.650, Y  +532.042, Z    +0.000, E1   -45.233, E3 +343587.748}
SPL {X  -165.650, Y  +537.290, Z    +0.000, E1   -45.204, E3 +343598.589}
SPL {X  -165.650, Y  +544.196, Z    +0.000, E1   -45.432, E3 +343611.263}
SPL {X  -165.650, Y  +548.678, Z    +0.000, E1   -45.162, E3 +343621.827}
SPL {X  -165.650, Y  +554.600, Z    +0.000, E1   -45.345, E3 +343632.804}
SPL {X  -165.650, Y  +559.896, Z    +0.000, E1   -45.150, E3 +343644.659}
SPL {X  -165.650, Y  +566.830, Z    +0.000, E1   -45.346, E3 +343657.640}
SPL {X  -165.650, Y  +573.074, Z    +0.000, E1   -45.379, E3 +343669.970}
SPL {X  -165.650, Y  +579.360, Z    +0.000, E1   -45.300, E3 +343683.255}
SPL {X  -165.650, Y  +584.577, Z    +0.000, E1   -45.167, E3 +343694.479}
SPL {X  -165.650, Y  +590.060, Z    +0.000, E1   -45.221, E3 +343705.370}
SPL {X  -165.650, Y  +596.611, Z    +0.000, E1   -45.390, E3 +343717.606}
SPL {X  -165.650, Y  +603.637, Z    +0.000, E1   -45.296, E3 +343732.525}
SPL {X  -165.650, Y  +610.850, Z    +0.000, E1   -45.208, E3 +343747.533}
SPL {X  -165.650, Y  +617.450, Z    +0.000, E1   -45.402, E3 +343759.735}
SPL {X  -165.650, Y  +622.720, Z    +0.000, E1   -45.272, E3 +343771.133}
SPL {X  -165.650, Y  +627.828, Z    +0.000, E1   -45.174, E3 +343782.090}
SPL {X  -165.650, Y  +634.620, Z    +0.000, E1   -45.438, E3 +343794.295}
SPL {X  -165.650, Y  +640.808, Z    +0.000, E1   -45.294, E3 +343807.670}
SPL {X  -165.650, Y  +646.552, Z    +0.000, E1   -45.137, E3 +343820.194}
SPL {X  -165.650, Y  +652.431, Z    +0.000, E1   -45.333, E3 +343830.949}
SPL {X  -165.650, Y  +657.443, Z    +0.000, E1   -45.316, E3 +343841.205}
SPL {X  -165.650, Y  +662.999, Z    +0.000, E1   -45.214, E3 +343853.077}
SPL {X  -165.650, Y  +668.737, Z    +0.000, E1   -45.236, E3 +343864.592}
SPL {X  -165.650, Y  +675.226, Z    +0.000, E1   -45.503, E3 +343876.095}
SPL {X  -165.597, Y  +679.672, Z    +0.000, E1   -45.206, E3 +343886.816}
SPL {X  -165.388, Y  +684.808, Z    +0.000, E1   -45.192, E3 +343897.324}
SPL {X  -165.020, Y  +689.938, Z    +0.000, E1   -45.107, E3 +343908.267}
SPL {X  -164.358, Y  +696.147, Z    +0.000, E1   -45.160, E3 +343920.532}
SPL {X  -163.631, Y  +701.286, Z    +0.000, E1   -44.994, E3 +343931.825}
SPL {X  -163.047, Y  +704.748, Z    +0.000, E1   -44.682, E3 +343940.648}
SPL {X  -161.884, Y  +710.619, Z    +0.000, E1   -44.738, E3 +343952.273}
SPL {X  -160.692, Y  +715.726, Z    +0.000, E1   -44.379, E3 +343964.596}
SPL {X  -159.384, Y  +720.631, Z    +0.000, E1   -44.155, E3 +343975.746}
SPL {X  -157.745, Y  +726.062, Z    +0.000, E1   -43.902, E3 +343988.232}
SPL {X  -153.030, Y  +738.918, Z    +0.000, E1   -47.123, E3 +343995.835}
SPL {X  -145.149, Y  +755.323, Z    +0.000, E1   -51.167, E3 +344001.967}
SPL {X  -144.116, Y  +757.172, Z    +0.000, E1   -42.809, E3 +344068.517}
SPL {X  -127.227, Y  +781.582, Z    +0.000, E1   -46.780, E3 +344114.186}
ENDSPLINE

SPLINE
SPL {X  -133.736, Y  +773.248, Z    +0.000, E1   -45.385, E3 +344192.229}
SPL {X  -160.761, Y  +715.447, Z    +0.000, E1   -23.748, E3 +344149.078}
SPL {X  -164.304, Y  +696.571, Z    +0.000, E1   -14.525, E3 +344154.302}
SPL {X  -165.374, Y  +685.052, Z    +0.000, E1    -8.166, E3 +344153.696}
SPL {X  -165.648, Y  +676.230, Z    +0.000, E1    -2.814, E3 +344152.847}
SPL {X  -165.650, Y  +670.481, Z    +0.000, E1    +1.454, E3 +344151.777}
SPL {X  -165.650, Y  +665.304, Z    +0.000, E1    +6.303, E3 +344150.279}
SPL {X  -165.650, Y  +660.688, Z    +0.000, E1   +11.392, E3 +344149.412}
SPL {X  -165.650, Y  +655.692, Z    +0.000, E1   +17.061, E3 +344148.834}
SPL {X  -165.650, Y  +646.511, Z    +0.000, E1   +26.434, E3 +344151.614}
SPL {X  -165.650, Y  +637.905, Z    +0.000, E1   +40.225, E3 +344139.739}
SPL {X  -165.650, Y  +607.385, Z    +0.000, E1   +51.775, E3 +344159.497}
SPL {X  -165.650, Y  +598.058, Z    +0.000, E1   +51.157, E3 +344172.958}
SPL {X  -165.650, Y  +553.219, Z    +0.000, E1   +52.865, E3 +344227.141}
ENDSPLINE

SPLINE
SPL {X  -165.650, Y  +569.883, Z    +0.000, E1   +45.183, E3 +344242.818}
ENDSPLINE

SPLINE
SPL {X  -165.650, Y  +564.081, Z    +0.000, E1   +45.208, E3 +344254.435}
SPL {X  -165.650, Y  +557.350, Z    +0.000, E1   +45.265, E3 +344267.872}
SPL {X  -165.650, Y  +549.414, Z    +0.000, E1   +45.294, E3 +344283.774}
SPL {X  -165.650, Y  +542.958, Z    +0.000, E1   +45.131, E3 +344297.777}
SPL {X  -165.650, Y  +535.288, Z    +0.000, E1   +45.332, E3 +344312.217}
SPL {X  -165.650, Y  +528.026, Z    +0.000, E1   +45.173, E3 +344327.876}
SPL {X  -165.650, Y  +520.964, Z    +0.000, E1   +45.458, E3 +344340.381}
SPL {X  -165.650, Y  +516.211, Z    +0.000, E1   +45.175, E3 +344351.724}
SPL {X  -165.650, Y  +511.047, Z    +0.000, E1   +45.193, E3 +344362.042}
SPL {X  -165.650, Y  +505.100, Z    +0.000, E1   +45.197, E3 +344374.246}
SPL {X  -165.650, Y  +499.646, Z    +0.000, E1   +44.886, E3 +344387.076}
ENDSPLINE

SPLINE
SPL {X  -165.650, Y  +514.834, Z    +0.000, E1   +36.829, E3 +344399.842}
ENDSPLINE

SPLINE
SPL {X  -165.650, Y  +506.421, Z    +0.000, E1   +37.886, E3 +344415.954}
SPL {X  -165.650, Y  +499.917, Z    +0.000, E1   +38.752, E3 +344427.415}
SPL {X  -165.650, Y  +493.826, Z    +0.000, E1   +39.521, E3 +344438.169}
SPL {X  -165.650, Y  +487.003, Z    +0.000, E1   +40.380, E3 +344449.623}
SPL {X  -165.650, Y  +478.382, Z    +0.000, E1   +41.628, E3 +344462.536}
SPL {X  -165.650, Y  +472.112, Z    +0.000, E1   +42.202, E3 +344473.274}
SPL {X  -165.650, Y  +466.741, Z    +0.000, E1   +42.890, E3 +344481.195}
SPL {X  -165.650, Y  +458.202, Z    +0.000, E1   +44.020, E3 +344492.983}
SPL {X  -165.650, Y  +449.099, Z    +0.000, E1   +44.871, E3 +344506.945}
SPL {X  -165.650, Y  +442.120, Z    +0.000, E1   +45.313, E3 +344518.497}
SPL {X  -165.650, Y  +436.063, Z    +0.000, E1   +44.972, E3 +344533.082}
SPL {X  -165.650, Y  +427.943, Z    +0.000, E1   +45.362, E3 +344547.119}
SPL {X  -165.650, Y  +422.523, Z    +0.000, E1   +45.103, E3 +344559.797}
SPL {X  -165.650, Y  +415.564, Z    +0.000, E1   +45.195, E3 +344573.336}
SPL {X  -165.650, Y  +410.687, Z    +0.000, E1   +44.955, E3 +344584.652}
SPL {X  -165.650, Y  +405.522, Z    +0.000, E1   +45.119, E3 +344594.212}
SPL {X  -165.650, Y  +399.216, Z    +0.000, E1   +45.246, E3 +344606.406}
SPL {X  -165.650, Y  +391.618, Z    +0.000, E1   +45.037, E3 +344623.184}
SPL {X  -165.650, Y  +383.700, Z    +0.000, E1   +45.345, E3 +344637.311}
SPL {X  -165.650, Y  +379.225, Z    +0.000, E1   +45.073, E3 +344648.000}
SPL {X  -165.591, Y  +374.097, Z    +0.000, E1   +45.069, E3 +344658.481}
SPL {X  -165.372, Y  +368.914, Z    +0.000, E1   +45.103, E3 +344668.841}
SPL {X  -164.987, Y  +363.696, Z    +0.000, E1   +45.006, E3 +344680.064}
SPL {X  -164.256, Y  +357.053, Z    +0.000, E1   +44.969, E3 +344693.867}
SPL {X  -163.441, Y  +351.538, Z    +0.000, E1   +44.749, E3 +344706.230}
SPL {X  -162.419, Y  +345.942, Z    +0.000, E1   +44.540, E3 +344718.962}
SPL {X  -161.210, Y  +340.404, Z    +0.000, E1   +44.250, E3 +344731.787}
SPL {X  -159.961, Y  +335.460, Z    +0.000, E1   +44.205, E3 +344742.150}
SPL {X  -158.595, Y  +330.672, Z    +0.000, E1   +43.797, E3 +344754.128}
SPL {X  -156.695, Y  +324.773, Z    +0.000, E1   +43.987, E3 +344765.025}
SPL {X  -148.318, Y  +304.733, Z    +0.000, E1   +49.897, E3 +344770.262}
SPL {X  -138.435, Y  +287.529, Z    +0.000, E1   +45.834, E3 +344835.586}
SPL {X  -134.645, Y  +282.008, Z    +0.000, E1   +45.207, E3 +344865.242}
ENDSPLINE

SPLINE
SPL {X  -154.915, Y  +319.839, Z    +0.000, E1   +31.584, E3 +344924.761}
SPL {X  -161.387, Y  +341.161, Z    +0.000, E1   +22.590, E3 +344938.607}
SPL {X  -164.566, Y  +359.576, Z    +0.000, E1   +13.425, E3 +344917.200}
SPL {X  -165.355, Y  +368.611, Z    +0.000, E1    +8.407, E3 +344920.781}
SPL {X  -165.614, Y  +375.050, Z    +0.000, E1    +4.520, E3 +344922.085}
SPL {X  -165.650, Y  +379.271, Z    +0.000, E1    +1.752, E3 +344919.107}
SPL {X  -165.650, Y  +382.603, Z    +0.000, E1    -0.657, E3 +344920.314}
SPL {X  -165.650, Y  +386.866, Z    +0.000, E1    -4.337, E3 +344919.580}
SPL {X  -165.650, Y  +394.200, Z    +0.000, E1   -11.943, E3 +344917.347}
SPL {X  -165.650, Y  +405.401, Z    +0.000, E1   -24.512, E3 +344917.168}
SPL {X  -165.650, Y  +418.038, Z    +0.000, E1   -38.688, E3 +344913.395}
SPL {X  -165.650, Y  +461.620, Z    +0.000, E1   -55.594, E3 +344933.574}
SPL {X  -165.650, Y  +498.574, Z    +0.000, E1   -52.082, E3 +344994.599}
ENDSPLINE

SPLINE
SPL {X  -165.650, Y  +483.168, Z    +0.000, E1   -45.573, E3 +345005.256}
ENDSPLINE

SPLINE
SPL {X  -165.650, Y  +487.615, Z    +0.000, E1   -45.254, E3 +345016.277}
SPL {X  -165.650, Y  +493.602, Z    +0.000, E1   -45.283, E3 +345028.117}
SPL {X  -165.650, Y  +498.857, Z    +0.000, E1   -45.339, E3 +345038.461}
SPL {X  -165.650, Y  +504.159, Z    +0.000, E1   -45.384, E3 +345048.856}
SPL {X  -165.650, Y  +509.628, Z    +0.000, E1   -45.217, E3 +345061.039}
SPL {X  -165.650, Y  +516.157, Z    +0.000, E1   -45.240, E3 +345074.074}
SPL {X  -165.650, Y  +521.049, Z    +0.000, E1   -45.236, E3 +345084.027}
SPL {X  -165.650, Y  +527.050, Z    +0.000, E1   -45.345, E3 +345095.523}
SPL {X  -165.650, Y  +532.042, Z    +0.000, E1   -45.233, E3 +345106.267}
SPL {X  -165.650, Y  +537.290, Z    +0.000, E1   -45.204, E3 +345117.107}
SPL {X  -165.650, Y  +544.196, Z    +0.000, E1   -45.432, E3 +345129.782}
SPL {X  -165.650, Y  +548.678, Z    +0.000, E1   -45.162, E3 +345140.345}
SPL {X  -165.650, Y  +554.600, Z    +0.000, E1   -45.345, E3 +345151.323}
SPL {X  -165.650, Y  +559.896, Z    +0.000, E1   -45.150, E3 +345163.178}
SPL {X  -165.650, Y  +566.830, Z    +0.000, E1   -45.346, E3 +345176.158}
SPL {X  -165.650, Y  +573.074, Z    +0.000, E1   -45.379, E3 +345188.489}
SPL {X  -165.650, Y  +579.360, Z    +0.000, E1   -45.300, E3 +345201.774}
SPL {X  -165.650, Y  +584.577, Z    +0.000, E1   -45.167, E3 +345212.997}
SPL {X  -165.650, Y  +590.060, Z    +0.000, E1   -45.221, E3 +345223.888}
SPL {X  -165.650, Y  +596.611, Z    +0.000, E1   -45.390, E3 +345236.124}
SPL {X  -165.650, Y  +603.637, Z    +0.000, E1   -45.296, E3 +345251.043}
SPL {X  -165.650, Y  +610.850, Z    +0.000, E1   -45.208, E3 +345266.051}
SPL {X  -165.650, Y  +617.450, Z    +0.000, E1   -45.402, E3 +345278.254}
SPL {X  -165.650, Y  +622.720, Z    +0.000, E1   -45.272, E3 +345289.651}
SPL {X  -165.650, Y  +627.828, Z    +0.000, E1   -45.174, E3 +345300.608}
SPL {X  -165.650, Y  +634.620, Z    +0.000, E1   -45.438, E3 +345312.814}
SPL {X  -165.650, Y  +640.808, Z    +0.000, E1   -45.294, E3 +345326.188}
SPL {X  -165.650, Y  +646.552, Z    +0.000, E1   -45.137, E3 +345338.713}
SPL {X  -165.650, Y  +652.431, Z    +0.000, E1   -45.333, E3 +345349.467}
SPL {X  -165.650, Y  +657.443, Z    +0.000, E1   -45.316, E3 +345359.723}
SPL {X  -165.650, Y  +662.999, Z    +0.000, E1   -45.214, E3 +345371.595}
SPL {X  -165.650, Y  +668.737, Z    +0.000, E1   -45.236, E3 +345383.110}
SPL {X  -165.650, Y  +675.226, Z    +0.000, E1   -45.503, E3 +345394.614}
SPL {X  -165.597, Y  +679.672, Z    +0.000, E1   -45.206, E3 +345405.335}
SPL {X  -165.388, Y  +684.808, Z    +0.000, E1   -45.192, E3 +345415.842}
SPL {X  -165.020, Y  +689.938, Z    +0.000, E1   -45.107, E3 +345426.785}
SPL {X  -164.358, Y  +696.147, Z    +0.000, E1   -45.160, E3 +345439.051}
SPL {X  -163.631, Y  +701.286, Z    +0.000, E1   -44.994, E3 +345450.343}
SPL {X  -163.047, Y  +704.748, Z    +0.000, E1   -44.682, E3 +345459.167}
SPL {X  -161.884, Y  +710.619, Z    +0.000, E1   -44.738, E3 +345470.792}
SPL {X  -160.692, Y  +715.726, Z    +0.000, E1   -44.379, E3 +345483.114}
SPL {X  -159.384, Y  +720.631, Z    +0.000, E1   -44.155, E3 +345494.264}
SPL {X  -157.745, Y  +726.062, Z    +0.000, E1   -43.902, E3 +345506.751}
SPL {X  -153.030, Y  +738.918, Z    +0.000, E1   -47.123, E3 +345514.353}
SPL {X  -145.149, Y  +755.323, Z    +0.000, E1   -51.167, E3 +345520.485}
SPL {X  -144.116, Y  +757.172, Z    +0.000, E1   -42.809, E3 +345587.035}
SPL {X  -127.227, Y  +781.582, Z    +0.000, E1   -46.780, E3 +345632.705}
ENDSPLINE

SPLINE
SPL {X  -133.736, Y  +773.248, Z    +0.000, E1   -45.385, E3 +345710.747}
SPL {X  -160.761, Y  +715.447, Z    +0.000, E1   -23.748, E3 +345667.597}
SPL {X  -164.304, Y  +696.571, Z    +0.000, E1   -14.525, E3 +345672.821}
SPL {X  -165.374, Y  +685.052, Z    +0.000, E1    -8.166, E3 +345672.215}
SPL {X  -165.648, Y  +676.230, Z    +0.000, E1    -2.814, E3 +345671.366}
SPL {X  -165.650, Y  +670.481, Z    +0.000, E1    +1.454, E3 +345670.295}
SPL {X  -165.650, Y  +665.304, Z    +0.000, E1    +6.303, E3 +345668.797}
SPL {X  -165.650, Y  +660.688, Z    +0.000, E1   +11.392, E3 +345667.930}
SPL {X  -165.650, Y  +655.692, Z    +0.000, E1   +17.061, E3 +345667.353}
SPL {X  -165.650, Y  +646.511, Z    +0.000, E1   +26.434, E3 +345670.133}
SPL {X  -165.650, Y  +637.905, Z    +0.000, E1   +40.225, E3 +345658.257}
SPL {X  -165.650, Y  +607.385, Z    +0.000, E1   +51.775, E3 +345678.015}
SPL {X  -165.650, Y  +598.058, Z    +0.000, E1   +51.157, E3 +345691.477}
SPL {X  -165.650, Y  +553.219, Z    +0.000, E1   +52.865, E3 +345745.659}
ENDSPLINE

SPLINE
SPL {X  -165.650, Y  +569.883, Z    +0.000, E1   +45.183, E3 +345761.336}
ENDSPLINE

SPLINE
SPL {X  -165.650, Y  +564.081, Z    +0.000, E1   +45.208, E3 +345772.954}
SPL {X  -165.650, Y  +557.350, Z    +0.000, E1   +45.265, E3 +345786.391}
SPL {X  -165.650, Y  +549.414, Z    +0.000, E1   +45.294, E3 +345802.293}
SPL {X  -165.650, Y  +542.958, Z    +0.000, E1   +45.131, E3 +345816.295}
SPL {X  -165.650, Y  +535.288, Z    +0.000, E1   +45.332, E3 +345830.736}
SPL {X  -165.650, Y  +528.026, Z    +0.000, E1   +45.173, E3 +345846.394}
SPL {X  -165.650, Y  +520.964, Z    +0.000, E1   +45.458, E3 +345858.899}
SPL {X  -165.650, Y  +516.211, Z    +0.000, E1   +45.175, E3 +345870.242}
SPL {X  -165.650, Y  +511.047, Z    +0.000, E1   +45.193, E3 +345880.561}
SPL {X  -165.650, Y  +505.100, Z    +0.000, E1   +45.197, E3 +345892.764}
SPL {X  -165.650, Y  +499.646, Z    +0.000, E1   +44.886, E3 +345905.594}
ENDSPLINE

SPLINE
SPL {X  -165.650, Y  +514.834, Z    +0.000, E1   +36.829, E3 +345918.360}
ENDSPLINE

SPLINE
SPL {X  -165.650, Y  +506.421, Z    +0.000, E1   +37.886, E3 +345934.472}
SPL {X  -165.650, Y  +499.917, Z    +0.000, E1   +38.752, E3 +345945.933}
SPL {X  -165.650, Y  +493.826, Z    +0.000, E1   +39.521, E3 +345956.687}
SPL {X  -165.650, Y  +487.003, Z    +0.000, E1   +40.380, E3 +345968.142}
SPL {X  -165.650, Y  +478.382, Z    +0.000, E1   +41.628, E3 +345981.054}
SPL {X  -165.650, Y  +472.112, Z    +0.000, E1   +42.202, E3 +345991.793}
SPL {X  -165.650, Y  +466.741, Z    +0.000, E1   +42.890, E3 +345999.714}
SPL {X  -165.650, Y  +458.202, Z    +0.000, E1   +44.020, E3 +346011.502}
SPL {X  -165.650, Y  +449.099, Z    +0.000, E1   +44.871, E3 +346025.464}
SPL {X  -165.650, Y  +442.120, Z    +0.000, E1   +45.313, E3 +346037.016}
SPL {X  -165.650, Y  +436.063, Z    +0.000, E1   +44.972, E3 +346051.600}
SPL {X  -165.650, Y  +427.943, Z    +0.000, E1   +45.362, E3 +346065.637}
SPL {X  -165.650, Y  +422.523, Z    +0.000, E1   +45.103, E3 +346078.316}
SPL {X  -165.650, Y  +415.564, Z    +0.000, E1   +45.195, E3 +346091.855}
SPL {X  -165.650, Y  +410.687, Z    +0.000, E1   +44.955, E3 +346103.171}
SPL {X  -165.650, Y  +405.522, Z    +0.000, E1   +45.119, E3 +346112.731}
SPL {X  -165.650, Y  +399.216, Z    +0.000, E1   +45.246, E3 +346124.925}
SPL {X  -165.650, Y  +391.618, Z    +0.000, E1   +45.037, E3 +346141.703}
SPL {X  -165.650, Y  +383.700, Z    +0.000, E1   +45.345, E3 +346155.829}
SPL {X  -165.650, Y  +379.225, Z    +0.000, E1   +45.073, E3 +346166.519}
SPL {X  -165.591, Y  +374.097, Z    +0.000, E1   +45.069, E3 +346177.000}
SPL {X  -165.372, Y  +368.914, Z    +0.000, E1   +45.103, E3 +346187.359}
SPL {X  -164.987, Y  +363.696, Z    +0.000, E1   +45.006, E3 +346198.582}
SPL {X  -164.256, Y  +357.053, Z    +0.000, E1   +44.969, E3 +346212.385}
SPL {X  -163.441, Y  +351.538, Z    +0.000, E1   +44.749, E3 +346224.749}
SPL {X  -162.419, Y  +345.942, Z    +0.000, E1   +44.540, E3 +346237.481}
SPL {X  -161.210, Y  +340.404, Z    +0.000, E1   +44.250, E3 +346250.305}
SPL {X  -159.961, Y  +335.460, Z    +0.000, E1   +44.205, E3 +346260.668}
SPL {X  -158.595, Y  +330.672, Z    +0.000, E1   +43.797, E3 +346272.647}
SPL {X  -156.695, Y  +324.773, Z    +0.000, E1   +43.987, E3 +346283.543}
SPL {X  -148.318, Y  +304.733, Z    +0.000, E1   +49.897, E3 +346288.780}
SPL {X  -138.435, Y  +287.529, Z    +0.000, E1   +45.834, E3 +346354.104}
SPL {X  -134.645, Y  +282.008, Z    +0.000, E1   +45.207, E3 +346383.761}
ENDSPLINE

SPLINE
SPL {X  -154.915, Y  +319.839, Z    +0.000, E1   +31.584, E3 +346443.280}
SPL {X  -161.387, Y  +341.161, Z    +0.000, E1   +22.590, E3 +346457.125}
SPL {X  -164.566, Y  +359.576, Z    +0.000, E1   +13.425, E3 +346435.719}
SPL {X  -165.355, Y  +368.611, Z    +0.000, E1    +8.407, E3 +346439.300}
SPL {X  -165.614, Y  +375.050, Z    +0.000, E1    +4.520, E3 +346440.603}
SPL {X  -165.650, Y  +379.271, Z    +0.000, E1    +1.752, E3 +346437.625}
SPL {X  -165.650, Y  +382.603, Z    +0.000, E1    -0.657, E3 +346438.833}
SPL {X  -165.650, Y  +386.866, Z    +0.000, E1    -4.337, E3 +346438.099}
SPL {X  -165.650, Y  +394.200, Z    +0.000, E1   -11.943, E3 +346435.866}
SPL {X  -165.650, Y  +405.401, Z    +0.000, E1   -24.512, E3 +346435.686}
SPL {X  -165.650, Y  +418.038, Z    +0.000, E1   -38.688, E3 +346431.913}
SPL {X  -165.650, Y  +461.620, Z    +0.000, E1   -55.594, E3 +346452.092}
SPL {X  -165.650, Y  +498.574, Z    +0.000, E1   -52.082, E3 +346513.117}
ENDSPLINE

SPLINE
SPL {X  -165.650, Y  +483.168, Z    +0.000, E1   -45.573, E3 +346523.774}
ENDSPLINE

SPLINE
SPL {X  -165.650, Y  +487.615, Z    +0.000, E1   -45.254, E3 +346534.796}
SPL {X  -165.650, Y  +493.602, Z    +0.000, E1   -45.283, E3 +346546.636}
SPL {X  -165.650, Y  +498.857, Z    +0.000, E1   -45.339, E3 +346556.980}
SPL {X  -165.650, Y  +504.159, Z    +0.000, E1   -45.384, E3 +346567.374}
SPL {X  -165.650, Y  +509.628, Z    +0.000, E1   -45.217, E3 +346579.557}
SPL {X  -165.650, Y  +516.157, Z    +0.000, E1   -45.240, E3 +346592.593}
SPL {X  -165.650, Y  +521.049, Z    +0.000, E1   -45.236, E3 +346602.546}
SPL {X  -165.650, Y  +527.050, Z    +0.000, E1   -45.345, E3 +346614.042}
SPL {X  -165.650, Y  +532.042, Z    +0.000, E1   -45.233, E3 +346624.785}
SPL {X  -165.650, Y  +537.290, Z    +0.000, E1   -45.204, E3 +346635.626}
SPL {X  -165.650, Y  +544.196, Z    +0.000, E1   -45.432, E3 +346648.300}
SPL {X  -165.650, Y  +548.678, Z    +0.000, E1   -45.162, E3 +346658.864}
SPL {X  -165.650, Y  +554.600, Z    +0.000, E1   -45.345, E3 +346669.841}
SPL {X  -165.650, Y  +559.896, Z    +0.000, E1   -45.150, E3 +346681.696}
SPL {X  -165.650, Y  +566.830, Z    +0.000, E1   -45.346, E3 +346694.677}
SPL {X  -165.650, Y  +573.074, Z    +0.000, E1   -45.379, E3 +346707.007}
SPL {X  -165.650, Y  +579.360, Z    +0.000, E1   -45.300, E3 +346720.292}
SPL {X  -165.650, Y  +584.577, Z    +0.000, E1   -45.167, E3 +346731.516}
SPL {X  -165.650, Y  +590.060, Z    +0.000, E1   -45.221, E3 +346742.407}
SPL {X  -165.650, Y  +596.611, Z    +0.000, E1   -45.390, E3 +346754.643}
SPL {X  -165.650, Y  +603.637, Z    +0.000, E1   -45.296, E3 +346769.562}
SPL {X  -165.650, Y  +610.850, Z    +0.000, E1   -45.208, E3 +346784.570}
SPL {X  -165.650, Y  +617.450, Z    +0.000, E1   -45.402, E3 +346796.772}
SPL {X  -165.650, Y  +622.720, Z    +0.000, E1   -45.272, E3 +346808.170}
SPL {X  -165.650, Y  +627.828, Z    +0.000, E1   -45.174, E3 +346819.127}
SPL {X  -165.650, Y  +634.620, Z    +0.000, E1   -45.438, E3 +346831.332}
SPL {X  -165.650, Y  +640.808, Z    +0.000, E1   -45.294, E3 +346844.707}
SPL {X  -165.650, Y  +646.552, Z    +0.000, E1   -45.137, E3 +346857.231}
SPL {X  -165.650, Y  +652.431, Z    +0.000, E1   -45.333, E3 +346867.986}
SPL {X  -165.650, Y  +657.443, Z    +0.000, E1   -45.316, E3 +346878.242}
SPL {X  -165.650, Y  +662.999, Z    +0.000, E1   -45.214, E3 +346890.114}
SPL {X  -165.650, Y  +668.737, Z    +0.000, E1   -45.236, E3 +346901.629}
SPL {X  -165.650, Y  +675.226, Z    +0.000, E1   -45.503, E3 +346913.132}
SPL {X  -165.597, Y  +679.672, Z    +0.000, E1   -45.206, E3 +346923.853}
SPL {X  -165.388, Y  +684.808, Z    +0.000, E1   -45.192, E3 +346934.361}
SPL {X  -165.020, Y  +689.938, Z    +0.000, E1   -45.107, E3 +346945.304}
SPL {X  -164.358, Y  +696.147, Z    +0.000, E1   -45.160, E3 +346957.570}
SPL {X  -163.631, Y  +701.286, Z    +0.000, E1   -44.994, E3 +346968.862}
SPL {X  -163.047, Y  +704.748, Z    +0.000, E1   -44.682, E3 +346977.685}
SPL {X  -161.884, Y  +710.619, Z    +0.000, E1   -44.738, E3 +346989.310}
SPL {X  -160.692, Y  +715.726, Z    +0.000, E1   -44.379, E3 +347001.633}
SPL {X  -159.384, Y  +720.631, Z    +0.000, E1   -44.155, E3 +347012.783}
SPL {X  -157.745, Y  +726.062, Z    +0.000, E1   -43.902, E3 +347025.269}
SPL {X  -153.030, Y  +738.918, Z    +0.000, E1   -47.123, E3 +347032.872}
SPL {X  -145.149, Y  +755.323, Z    +0.000, E1   -51.167, E3 +347039.004}
SPL {X  -144.116, Y  +757.172, Z    +0.000, E1   -42.809, E3 +347105.554}
SPL {X  -127.227, Y  +781.582, Z    +0.000, E1   -46.780, E3 +347151.223}
ENDSPLINE

SPLINE
SPL {X  -133.736, Y  +773.248, Z    +0.000, E1   -45.385, E3 +347229.266}
SPL {X  -160.761, Y  +715.447, Z    +0.000, E1   -23.748, E3 +347186.115}
SPL {X  -164.304, Y  +696.571, Z    +0.000, E1   -14.525, E3 +347191.339}
SPL {X  -165.374, Y  +685.052, Z    +0.000, E1    -8.166, E3 +347190.733}
SPL {X  -165.648, Y  +676.230, Z    +0.000, E1    -2.814, E3 +347189.884}
SPL {X  -165.650, Y  +670.481, Z    +0.000, E1    +1.454, E3 +347188.814}
SPL {X  -165.650, Y  +665.304, Z    +0.000, E1    +6.303, E3 +347187.316}
SPL {X  -165.650, Y  +660.688, Z    +0.000, E1   +11.392, E3 +347186.449}
SPL {X  -165.650, Y  +655.692, Z    +0.000, E1   +17.061, E3 +347185.871}
SPL {X  -165.650, Y  +646.511, Z    +0.000, E1   +26.434, E3 +347188.651}
SPL {X  -165.650, Y  +637.905, Z    +0.000, E1   +40.225, E3 +347176.776}
SPL {X  -165.650, Y  +607.385, Z    +0.000, E1   +51.775, E3 +347196.534}
SPL {X  -165.650, Y  +598.058, Z    +0.000, E1   +51.157, E3 +347209.995}
SPL {X  -165.650, Y  +553.219, Z    +0.000, E1   +52.865, E3 +347264.178}
ENDSPLINE

SPLINE
SPL {X  -165.650, Y  +569.883, Z    +0.000, E1   +45.183, E3 +347279.855}
ENDSPLINE

SPLINE
SPL {X  -165.650, Y  +564.081, Z    +0.000, E1   +45.208, E3 +347291.472}
SPL {X  -165.650, Y  +557.350, Z    +0.000, E1   +45.265, E3 +347304.910}
SPL {X  -165.650, Y  +549.414, Z    +0.000, E1   +45.294, E3 +347320.811}
SPL {X  -165.650, Y  +542.958, Z    +0.000, E1   +45.131, E3 +347334.814}
SPL {X  -165.650, Y  +535.288, Z    +0.000, E1   +45.332, E3 +347349.254}
SPL {X  -165.650, Y  +528.026, Z    +0.000, E1   +45.173, E3 +347364.913}
SPL {X  -165.650, Y  +520.964, Z    +0.000, E1   +45.458, E3 +347377.418}
SPL {X  -165.650, Y  +516.211, Z    +0.000, E1   +45.175, E3 +347388.761}
SPL {X  -165.650, Y  +511.047, Z    +0.000, E1   +45.193, E3 +347399.079}
SPL {X  -165.650, Y  +505.100, Z    +0.000, E1   +45.197, E3 +347411.283}
SPL {X  -165.650, Y  +499.646, Z    +0.000, E1   +44.886, E3 +347424.113}
ENDSPLINE

SPLINE
SPL {X  -165.650, Y  +514.834, Z    +0.000, E1   +36.829, E3 +347436.879}
ENDSPLINE

SPLINE
SPL {X  -165.650, Y  +506.421, Z    +0.000, E1   +37.886, E3 +347452.991}
SPL {X  -165.650, Y  +499.917, Z    +0.000, E1   +38.752, E3 +347464.452}
SPL {X  -165.650, Y  +493.826, Z    +0.000, E1   +39.521, E3 +347475.206}
SPL {X  -165.650, Y  +487.003, Z    +0.000, E1   +40.380, E3 +347486.660}
SPL {X  -165.650, Y  +478.382, Z    +0.000, E1   +41.628, E3 +347499.573}
SPL {X  -165.650, Y  +472.112, Z    +0.000, E1   +42.202, E3 +347510.311}
SPL {X  -165.650, Y  +466.741, Z    +0.000, E1   +42.890, E3 +347518.232}
SPL {X  -165.650, Y  +458.202, Z    +0.000, E1   +44.020, E3 +347530.020}
SPL {X  -165.650, Y  +449.099, Z    +0.000, E1   +44.871, E3 +347543.982}
SPL {X  -165.650, Y  +442.120, Z    +0.000, E1   +45.313, E3 +347555.534}
SPL {X  -165.650, Y  +436.063, Z    +0.000, E1   +44.972, E3 +347570.119}
SPL {X  -165.650, Y  +427.943, Z    +0.000, E1   +45.362, E3 +347584.156}
SPL {X  -165.650, Y  +422.523, Z    +0.000, E1   +45.103, E3 +347596.834}
SPL {X  -165.650, Y  +415.564, Z    +0.000, E1   +45.195, E3 +347610.373}
SPL {X  -165.650, Y  +410.687, Z    +0.000, E1   +44.955, E3 +347621.689}
SPL {X  -165.650, Y  +405.522, Z    +0.000, E1   +45.119, E3 +347631.249}
SPL {X  -165.650, Y  +399.216, Z    +0.000, E1   +45.246, E3 +347643.443}
SPL {X  -165.650, Y  +391.618, Z    +0.000, E1   +45.037, E3 +347660.221}
SPL {X  -165.650, Y  +383.700, Z    +0.000, E1   +45.345, E3 +347674.348}
SPL {X  -165.650, Y  +379.225, Z    +0.000, E1   +45.073, E3 +347685.037}
SPL {X  -165.591, Y  +374.097, Z    +0.000, E1   +45.069, E3 +347695.518}
SPL {X  -165.372, Y  +368.914, Z    +0.000, E1   +45.103, E3 +347705.878}
SPL {X  -164.987, Y  +363.696, Z    +0.000, E1   +45.006, E3 +347717.101}
SPL {X  -164.256, Y  +357.053, Z    +0.000, E1   +44.969, E3 +347730.904}
SPL {X  -163.441, Y  +351.538, Z    +0.000, E1   +44.749, E3 +347743.267}
SPL {X  -162.419, Y  +345.942, Z    +0.000, E1   +44.540, E3 +347755.999}
SPL {X  -161.210, Y  +340.404, Z    +0.000, E1   +44.250, E3 +347768.824}
SPL {X  -159.961, Y  +335.460, Z    +0.000, E1   +44.205, E3 +347779.187}
SPL {X  -158.595, Y  +330.672, Z    +0.000, E1   +43.797, E3 +347791.165}
SPL {X  -156.695, Y  +324.773, Z    +0.000, E1   +43.987, E3 +347802.062}
SPL {X  -148.318, Y  +304.733, Z    +0.000, E1   +49.897, E3 +347807.299}
SPL {X  -138.435, Y  +287.529, Z    +0.000, E1   +45.834, E3 +347872.623}
SPL {X  -134.645, Y  +282.008, Z    +0.000, E1   +45.207, E3 +347902.279}
ENDSPLINE

SPLINE
SPL {X  -154.915, Y  +319.839, Z    +0.000, E1   +31.584, E3 +347961.798}
SPL {X  -161.387, Y  +341.161, Z    +0.000, E1   +22.590, E3 +347975.644}
SPL {X  -164.566, Y  +359.576, Z    +0.000, E1   +13.425, E3 +347954.237}
SPL {X  -165.355, Y  +368.611, Z    +0.000, E1    +8.407, E3 +347957.818}
SPL {X  -165.614, Y  +375.050, Z    +0.000, E1    +4.520, E3 +347959.122}
SPL {X  -165.650, Y  +379.847, Z    +0.000, E1    +1.364, E3 +347957.471}
SPL {X  -165.650, Y  +384.387, Z    +0.000, E1    -2.084, E3 +347956.453}
SPL {X  -165.650, Y  +387.977, Z    +0.000, E1    -5.454, E3 +347956.938}
SPL {X  -165.650, Y  +392.464, Z    +0.000, E1   -10.170, E3 +347954.621}
SPL {X  -165.650, Y  +397.361, Z    +0.000, E1   -15.736, E3 +347953.953}
SPL {X  -165.650, Y  +404.553, Z    +0.000, E1   -23.488, E3 +347954.729}
SPL {X  -165.650, Y  +415.773, Z    +0.000, E1   -36.308, E3 +347950.881}
SPL {X  -165.650, Y  +461.620, Z    +0.000, E1   -55.594, E3 +347970.611}
SPL {X  -165.650, Y  +498.574, Z    +0.000, E1   -52.082, E3 +348031.636}
ENDSPLINE

SPLINE
SPL {X  -165.650, Y  +483.168, Z    +0.000, E1   -45.573, E3 +348042.293}
ENDSPLINE

SPLINE
SPL {X  -165.650, Y  +487.615, Z    +0.000, E1   -45.254, E3 +348053.314}
SPL {X  -165.650, Y  +493.602, Z    +0.000, E1   -45.283, E3 +348065.154}
SPL {X  -165.650, Y  +498.857, Z    +0.000, E1   -45.339, E3 +348075.498}
SPL {X  -165.650, Y  +505.115, Z    +0.000, E1   -45.299, E3 +348088.446}
SPL {X  -165.650, Y  +510.931, Z    +0.000, E1   -45.250, E3 +348100.437}
SPL {X  -165.650, Y  +516.157, Z    +0.000, E1   -45.240, E3 +348111.111}
SPL {X  -165.650, Y  +521.049, Z    +0.000, E1   -45.236, E3 +348121.064}
SPL {X  -165.650, Y  +527.050, Z    +0.000, E1   -45.345, E3 +348132.560}
SPL {X  -165.650, Y  +532.042, Z    +0.000, E1   -45.233, E3 +348143.304}
SPL {X  -165.650, Y  +537.290, Z    +0.000, E1   -45.204, E3 +348154.145}
SPL {X  -165.650, Y  +544.196, Z    +0.000, E1   -45.432, E3 +348166.819}
SPL {X  -165.650, Y  +548.678, Z    +0.000, E1   -45.162, E3 +348177.383}
SPL {X  -165.650, Y  +554.600, Z    +0.000, E1   -45.345, E3 +348188.360}
SPL {X  -165.650, Y  +559.896, Z    +0.000, E1   -45.150, E3 +348200.215}
SPL {X  -165.650, Y  +566.830, Z    +0.000, E1   -45.346, E3 +348213.195}
SPL {X  -165.650, Y  +573.074, Z    +0.000, E1   -45.379, E3 +348225.526}
SPL {X  -165.650, Y  +577.292, Z    +0.000, E1   -45.246, E3 +348234.790}
SPL {X  -165.650, Y  +583.131, Z    +0.000, E1   -45.255, E3 +348246.731}
SPL {X  -165.650, Y  +590.060, Z    +0.000, E1   -45.221, E3 +348260.925}
SPL {X  -165.650, Y  +596.611, Z    +0.000, E1   -45.390, E3 +348273.161}
SPL {X  -165.650, Y  +603.637, Z    +0.000, E1   -45.296, E3 +348288.080}
SPL {X  -165.650, Y  +610.850, Z    +0.000, E1   -45.208, E3 +348303.088}
SPL {X  -165.650, Y  +617.450, Z    +0.000, E1   -45.402, E3 +348315.291}
SPL {X  -165.650, Y  +622.720, Z    +0.000, E1   -45.272, E3 +348326.689}
SPL {X  -165.650, Y  +627.828, Z    +0.000, E1   -45.174, E3 +348337.645}
SPL {X  -165.650, Y  +634.620, Z    +0.000, E1   -45.438, E3 +348349.851}
SPL {X  -165.650, Y  +640.808, Z    +0.000, E1   -45.294, E3 +348363.225}
SPL {X  -165.650, Y  +646.552, Z    +0.000, E1   -45.137, E3 +348375.750}
SPL {X  -165.650, Y  +652.431, Z    +0.000, E1   -45.333, E3 +348386.504}
SPL {X  -165.650, Y  +657.443, Z    +0.000, E1   -45.316, E3 +348396.760}
SPL {X  -165.650, Y  +662.999, Z    +0.000, E1   -45.214, E3 +348408.632}
SPL {X  -165.650, Y  +668.737, Z    +0.000, E1   -45.236, E3 +348420.147}
SPL {X  -165.650, Y  +675.226, Z    +0.000, E1   -45.503, E3 +348431.651}
SPL {X  -165.597, Y  +679.672, Z    +0.000, E1   -45.206, E3 +348442.372}
SPL {X  -165.388, Y  +684.808, Z    +0.000, E1   -45.192, E3 +348452.880}
SPL {X  -165.020, Y  +689.938, Z    +0.000, E1   -45.107, E3 +348463.822}
SPL {X  -164.358, Y  +696.147, Z    +0.000, E1   -45.160, E3 +348476.088}
SPL {X  -163.631, Y  +701.286, Z    +0.000, E1   -44.994, E3 +348487.380}
SPL {X  -163.047, Y  +704.748, Z    +0.000, E1   -44.682, E3 +348496.204}
SPL {X  -161.884, Y  +710.619, Z    +0.000, E1   -44.738, E3 +348507.829}
SPL {X  -160.692, Y  +715.726, Z    +0.000, E1   -44.379, E3 +348520.151}
SPL {X  -159.384, Y  +720.631, Z    +0.000, E1   -44.155, E3 +348531.301}
SPL {X  -157.745, Y  +726.062, Z    +0.000, E1   -43.902, E3 +348543.788}
SPL {X  -153.030, Y  +738.918, Z    +0.000, E1   -47.123, E3 +348551.390}
SPL {X  -145.149, Y  +755.323, Z    +0.000, E1   -51.167, E3 +348557.522}
SPL {X  -144.116, Y  +757.172, Z    +0.000, E1   -42.809, E3 +348624.072}
SPL {X  -127.227, Y  +781.582, Z    +0.000, E1   -46.780, E3 +348669.742}
ENDSPLINE

SPLINE
SPL {X  -133.736, Y  +773.248, Z    +0.000, E1   -45.385, E3 +348747.784}
SPL {X  -160.761, Y  +715.447, Z    +0.000, E1   -23.748, E3 +348704.634}
SPL {X  -164.304, Y  +696.571, Z    +0.000, E1   -14.525, E3 +348709.858}
SPL {X  -165.374, Y  +685.052, Z    +0.000, E1    -8.166, E3 +348709.252}
SPL {X  -165.648, Y  +676.230, Z    +0.000, E1    -2.814, E3 +348708.403}
SPL {X  -165.650, Y  +670.481, Z    +0.000, E1    +1.454, E3 +348707.332}
SPL {X  -165.650, Y  +665.304, Z    +0.000, E1    +6.303, E3 +348705.834}
SPL {X  -165.650, Y  +660.688, Z    +0.000, E1   +11.392, E3 +348704.967}
SPL {X  -165.650, Y  +655.692, Z    +0.000, E1   +17.061, E3 +348704.390}
SPL {X  -165.650, Y  +646.511, Z    +0.000, E1   +26.434, E3 +348707.170}
SPL {X  -165.650, Y  +637.905, Z    +0.000, E1   +40.225, E3 +348695.294}
SPL {X  -165.650, Y  +607.385, Z    +0.000, E1   +51.775, E3 +348715.052}
SPL {X  -165.650, Y  +598.058, Z    +0.000, E1   +51.157, E3 +348728.514}
SPL {X  -165.650, Y  +553.219, Z    +0.000, E1   +52.865, E3 +348782.696}
ENDSPLINE

SPLINE
SPL {X  -165.650, Y  +569.883, Z    +0.000, E1   +45.183, E3 +348798.373}
ENDSPLINE

SPLINE
SPL {X  -165.650, Y  +564.081, Z    +0.000, E1   +45.208, E3 +348809.991}
SPL {X  -165.650, Y  +557.350, Z    +0.000, E1   +45.265, E3 +348823.428}
SPL {X  -165.650, Y  +549.414, Z    +0.000, E1   +45.294, E3 +348839.330}
SPL {X  -165.650, Y  +542.958, Z    +0.000, E1   +45.131, E3 +348853.332}
SPL {X  -165.650, Y  +535.288, Z    +0.000, E1   +45.332, E3 +348867.773}
SPL {X  -165.650, Y  +528.026, Z    +0.000, E1   +45.173, E3 +348883.431}
SPL {X  -165.650, Y  +520.964, Z    +0.000, E1   +45.458, E3 +348895.936}
SPL {X  -165.650, Y  +516.211, Z    +0.000, E1   +45.175, E3 +348907.279}
SPL {X  -165.650, Y  +511.047, Z    +0.000, E1   +45.193, E3 +348917.598}
SPL {X  -165.650, Y  +505.100, Z    +0.000, E1   +45.197, E3 +348929.801}
SPL {X  -165.650, Y  +499.646, Z    +0.000, E1   +44.886, E3 +348942.631}
ENDSPLINE

SPLINE
SPL {X  -165.650, Y  +514.834, Z    +0.000, E1   +36.829, E3 +348955.397}
ENDSPLINE

SPLINE
SPL {X  -165.650, Y  +506.421, Z    +0.000, E1   +37.886, E3 +348971.509}
SPL {X  -165.650, Y  +499.917, Z    +0.000, E1   +38.752, E3 +348982.970}
SPL {X  -165.650, Y  +493.826, Z    +0.000, E1   +39.521, E3 +348993.724}
SPL {X  -165.650, Y  +487.003, Z    +0.000, E1   +40.380, E3 +349005.179}
SPL {X  -165.650, Y  +478.382, Z    +0.000, E1   +41.628, E3 +349018.091}
SPL {X  -165.650, Y  +472.112, Z    +0.000, E1   +42.202, E3 +349028.830}
SPL {X  -165.650, Y  +466.741, Z    +0.000, E1   +42.890, E3 +349036.751}
SPL {X  -165.650, Y  +458.202, Z    +0.000, E1   +44.020, E3 +349048.539}
SPL {X  -165.650, Y  +449.099, Z    +0.000, E1   +44.871, E3 +349062.501}
SPL {X  -165.650, Y  +442.120, Z    +0.000, E1   +45.313, E3 +349074.053}
SPL {X  -165.650, Y  +436.063, Z    +0.000, E1   +44.972, E3 +349088.637}
SPL {X  -165.650, Y  +427.943, Z    +0.000, E1   +45.362, E3 +349102.674}
SPL {X  -165.650, Y  +422.523, Z    +0.000, E1   +45.103, E3 +349115.353}
SPL {X  -165.650, Y  +415.564, Z    +0.000, E1   +45.195, E3 +349128.892}
SPL {X  -165.650, Y  +410.687, Z    +0.000, E1   +44.955, E3 +349140.208}
SPL {X  -165.650, Y  +405.522, Z    +0.000, E1   +45.119, E3 +349149.768}
SPL {X  -165.650, Y  +399.216, Z    +0.000, E1   +45.246, E3 +349161.962}
SPL {X  -165.650, Y  +391.618, Z    +0.000, E1   +45.037, E3 +349178.740}
SPL {X  -165.650, Y  +383.700, Z    +0.000, E1   +45.345, E3 +349192.866}
SPL {X  -165.650, Y  +379.225, Z    +0.000, E1   +45.073, E3 +349203.556}
SPL {X  -165.591, Y  +374.097, Z    +0.000, E1   +45.069, E3 +349214.037}
SPL {X  -165.372, Y  +368.914, Z    +0.000, E1   +45.103, E3 +349224.397}
SPL {X  -164.987, Y  +363.696, Z    +0.000, E1   +45.006, E3 +349235.620}
SPL {X  -164.256, Y  +357.053, Z    +0.000, E1   +44.969, E3 +349249.422}
SPL {X  -163.441, Y  +351.538, Z    +0.000, E1   +44.749, E3 +349261.786}
SPL {X  -162.419, Y  +345.942, Z    +0.000, E1   +44.540, E3 +349274.518}
SPL {X  -161.210, Y  +340.404, Z    +0.000, E1   +44.250, E3 +349287.342}
SPL {X  -159.961, Y  +335.460, Z    +0.000, E1   +44.205, E3 +349297.705}
SPL {X  -158.595, Y  +330.672, Z    +0.000, E1   +43.797, E3 +349309.684}
SPL {X  -156.695, Y  +324.773, Z    +0.000, E1   +43.987, E3 +349320.580}
SPL {X  -148.318, Y  +304.733, Z    +0.000, E1   +49.897, E3 +349325.817}
SPL {X  -138.435, Y  +287.529, Z    +0.000, E1   +45.834, E3 +349391.142}
SPL {X  -134.645, Y  +282.008, Z    +0.000, E1   +45.207, E3 +349420.798}
ENDSPLINE

SPLINE
SPL {X  -154.915, Y  +319.839, Z    +0.000, E1   +31.584, E3 +349480.317}
SPL {X  -161.387, Y  +341.161, Z    +0.000, E1   +22.590, E3 +349494.162}
SPL {X  -164.566, Y  +359.576, Z    +0.000, E1   +13.425, E3 +349472.756}
SPL {X  -165.355, Y  +368.611, Z    +0.000, E1    +8.407, E3 +349476.337}
SPL {X  -165.614, Y  +375.050, Z    +0.000, E1    +4.520, E3 +349477.640}
SPL {X  -165.650, Y  +379.271, Z    +0.000, E1    +1.752, E3 +349474.662}
SPL {X  -165.650, Y  +382.603, Z    +0.000, E1    -0.657, E3 +349475.870}
SPL {X  -165.650, Y  +386.866, Z    +0.000, E1    -4.337, E3 +349475.136}
SPL {X  -165.650, Y  +394.200, Z    +0.000, E1   -11.943, E3 +349472.903}
SPL {X  -165.650, Y  +405.401, Z    +0.000, E1   -24.512, E3 +349472.723}
SPL {X  -165.650, Y  +418.038, Z    +0.000, E1   -38.688, E3 +349468.950}
SPL {X  -165.650, Y  +461.620, Z    +0.000, E1   -55.594, E3 +349489.129}
SPL {X  -165.650, Y  +498.574, Z    +0.000, E1   -52.082, E3 +349550.154}
ENDSPLINE

SPLINE
SPL {X  -165.650, Y  +483.168, Z    +0.000, E1   -45.573, E3 +349560.811}
ENDSPLINE

SPLINE
SPL {X  -165.650, Y  +487.615, Z    +0.000, E1   -45.254, E3 +349571.833}
SPL {X  -165.650, Y  +493.602, Z    +0.000, E1   -45.283, E3 +349583.673}
SPL {X  -165.650, Y  +498.857, Z    +0.000, E1   -45.339, E3 +349594.017}
SPL {X  -165.650, Y  +504.159, Z    +0.000, E1   -45.384, E3 +349604.411}
SPL {X  -165.650, Y  +509.628, Z    +0.000, E1   -45.217, E3 +349616.595}
SPL {X  -165.650, Y  +516.157, Z    +0.000, E1   -45.240, E3 +349629.630}
SPL {X  -165.650, Y  +521.049, Z    +0.000, E1   -45.236, E3 +349639.583}
SPL {X  -165.650, Y  +527.050, Z    +0.000, E1   -45.345, E3 +349651.079}
SPL {X  -165.650, Y  +532.042, Z    +0.000, E1   -45.233, E3 +349661.822}
SPL {X  -165.650, Y  +537.290, Z    +0.000, E1   -45.204, E3 +349672.663}
SPL {X  -165.650, Y  +544.196, Z    +0.000, E1   -45.432, E3 +349685.337}
SPL {X  -165.650, Y  +548.678, Z    +0.000, E1   -45.162, E3 +349695.901}
SPL {X  -165.650, Y  +554.600, Z    +0.000, E1   -45.345, E3 +349706.878}
SPL {X  -165.650, Y  +559.896, Z    +0.000, E1   -45.150, E3 +349718.733}
SPL {X  -165.650, Y  +566.830, Z    +0.000, E1   -45.346, E3 +349731.714}
SPL {X  -165.650, Y  +573.074, Z    +0.000, E1   -45.379, E3 +349744.044}
SPL {X  -165.650, Y  +579.360, Z    +0.000, E1   -45.300, E3 +349757.330}
SPL {X  -165.650, Y  +584.577, Z    +0.000, E1   -45.167, E3 +349768.553}
SPL {X  -165.650, Y  +590.060, Z    +0.000, E1   -45.221, E3 +349779.444}
SPL {X  -165.650, Y  +596.611, Z    +0.000, E1   -45.390, E3 +349791.680}
SPL {X  -165.650, Y  +603.637, Z    +0.000, E1   -45.296, E3 +349806.599}
SPL {X  -165.650, Y  +610.850, Z    +0.000, E1   -45.208, E3 +349821.607}
SPL {X  -165.650, Y  +617.450, Z    +0.000, E1   -45.402, E3 +349833.809}
SPL {X  -165.650, Y  +622.720, Z    +0.000, E1   -45.272, E3 +349845.207}
SPL {X  -165.650, Y  +627.828, Z    +0.000, E1   -45.174, E3 +349856.164}
SPL {X  -165.650, Y  +634.620, Z    +0.000, E1   -45.438, E3 +349868.369}
SPL {X  -165.650, Y  +640.808, Z    +0.000, E1   -45.294, E3 +349881.744}
SPL {X  -165.650, Y  +646.552, Z    +0.000, E1   -45.137, E3 +349894.268}
SPL {X  -165.650, Y  +652.431, Z    +0.000, E1   -45.333, E3 +349905.023}
SPL {X  -165.650, Y  +657.443, Z    +0.000, E1   -45.316, E3 +349915.279}
SPL {X  -165.650, Y  +662.999, Z    +0.000, E1   -45.214, E3 +349927.151}
SPL {X  -165.650, Y  +668.737, Z    +0.000, E1   -45.236, E3 +349938.666}
SPL {X  -165.650, Y  +675.226, Z    +0.000, E1   -45.503, E3 +349950.169}
SPL {X  -165.597, Y  +679.672, Z    +0.000, E1   -45.206, E3 +349960.890}
SPL {X  -165.388, Y  +684.808, Z    +0.000, E1   -45.192, E3 +349971.398}
SPL {X  -165.020, Y  +689.938, Z    +0.000, E1   -45.107, E3 +349982.341}
SPL {X  -164.358, Y  +696.147, Z    +0.000, E1   -45.160, E3 +349994.607}
SPL {X  -163.631, Y  +701.286, Z    +0.000, E1   -44.994, E3 +350005.899}
SPL {X  -163.047, Y  +704.748, Z    +0.000, E1   -44.682, E3 +350014.722}
SPL {X  -161.884, Y  +710.619, Z    +0.000, E1   -44.738, E3 +350026.347}
SPL {X  -160.692, Y  +715.726, Z    +0.000, E1   -44.379, E3 +350038.670}
SPL {X  -159.384, Y  +720.631, Z    +0.000, E1   -44.155, E3 +350049.820}
SPL {X  -157.745, Y  +726.062, Z    +0.000, E1   -43.902, E3 +350062.306}
SPL {X  -153.030, Y  +738.918, Z    +0.000, E1   -47.123, E3 +350069.909}
SPL {X  -145.149, Y  +755.323, Z    +0.000, E1   -51.167, E3 +350076.041}
SPL {X  -143.038, Y  +759.047, Z    +0.000, E1   -43.157, E3 +350145.215}
SPL {X  -123.277, Y  +786.146, Z    +0.000, E1   -47.533, E3 +350201.270}
ENDSPLINE

SPLINE
SPL {X  -133.736, Y  +773.248, Z    +0.000, E1   -45.385, E3 +350266.303}
SPL {X  -160.761, Y  +715.447, Z    +0.000, E1   -23.748, E3 +350223.152}
SPL {X  -164.304, Y  +696.571, Z    +0.000, E1   -14.525, E3 +350228.376}
SPL {X  -165.498, Y  +682.585, Z    +0.000, E1    -6.769, E3 +350228.051}
SPL {X  -165.650, Y  +674.975, Z    +0.000, E1    -1.888, E3 +350226.409}
SPL {X  -165.650, Y  +671.520, Z    +0.000, E1    +0.682, E3 +350225.336}
SPL {X  -165.650, Y  +669.226, Z    +0.000, E1    +2.606, E3 +350226.470}
SPL {X  -165.650, Y  +665.304, Z    +0.000, E1    +6.303, E3 +350224.353}
SPL {X  -165.650, Y  +657.587, Z    +0.000, E1   +14.733, E3 +350223.127}
SPL {X  -165.650, Y  +646.511, Z    +0.000, E1   +26.434, E3 +350225.688}
SPL {X  -165.650, Y  +637.905, Z    +0.000, E1   +40.225, E3 +350213.813}
SPL {X  -165.650, Y  +607.385, Z    +0.000, E1   +51.775, E3 +350233.571}
SPL {X  -165.650, Y  +598.058, Z    +0.000, E1   +51.157, E3 +350247.032}
SPL {X  -165.650, Y  +553.656, Z    +0.000, E1   +53.998, E3 +350294.032}
SPL {X  -165.650, Y  +553.154, Z    +0.000, E1   +52.102, E3 +350305.559}
ENDSPLINE

SPLINE
SPL {X  -165.650, Y  +569.883, Z    +0.000, E1   +45.183, E3 +350316.892}
ENDSPLINE

SPLINE
SPL {X  -165.650, Y  +564.081, Z    +0.000, E1   +45.208, E3 +350328.509}
SPL {X  -165.650, Y  +557.350, Z    +0.000, E1   +45.265, E3 +350341.947}
SPL {X  -165.650, Y  +549.414, Z    +0.000, E1   +45.294, E3 +350357.849}
SPL {X  -165.650, Y  +542.958, Z    +0.000, E1   +45.131, E3 +350371.851}
SPL {X  -165.650, Y  +535.288, Z    +0.000, E1   +45.332, E3 +350386.291}
SPL {X  -165.650, Y  +528.026, Z    +0.000, E1   +45.173, E3 +350401.950}
SPL {X  -165.650, Y  +520.964, Z    +0.000, E1   +45.458, E3 +350414.455}
SPL {X  -165.650, Y  +516.211, Z    +0.000, E1   +45.175, E3 +350425.798}
SPL {X  -165.650, Y  +511.047, Z    +0.000, E1   +45.193, E3 +350436.116}
SPL {X  -165.650, Y  +505.100, Z    +0.000, E1   +45.197, E3 +350448.320}
SPL {X  -165.650, Y  +499.646, Z    +0.000, E1   +44.886, E3 +350461.150}
ENDSPLINE

SPLINE
SPL {X  -165.650, Y  +514.834, Z    +0.000, E1   +36.829, E3 +350473.916}
ENDSPLINE

SPLINE
SPL {X  -165.650, Y  +506.421, Z    +0.000, E1   +37.886, E3 +350490.028}
SPL {X  -165.650, Y  +499.917, Z    +0.000, E1   +38.752, E3 +350501.489}
SPL {X  -165.650, Y  +493.826, Z    +0.000, E1   +39.521, E3 +350512.243}
SPL {X  -165.650, Y  +487.003, Z    +0.000, E1   +40.380, E3 +350523.697}
SPL {X  -165.650, Y  +478.382, Z    +0.000, E1   +41.628, E3 +350536.610}
SPL {X  -165.650, Y  +472.112, Z    +0.000, E1   +42.202, E3 +350547.348}
SPL {X  -165.650, Y  +466.741, Z    +0.000, E1   +42.890, E3 +350555.269}
SPL {X  -165.650, Y  +458.202, Z    +0.000, E1   +44.020, E3 +350567.057}
SPL {X  -165.650, Y  +449.099, Z    +0.000, E1   +44.871, E3 +350581.019}
SPL {X  -165.650, Y  +442.120, Z    +0.000, E1   +45.313, E3 +350592.571}
SPL {X  -165.650, Y  +436.063, Z    +0.000, E1   +44.972, E3 +350607.156}
SPL {X  -165.650, Y  +427.943, Z    +0.000, E1   +45.362, E3 +350621.193}
SPL {X  -165.650, Y  +422.523, Z    +0.000, E1   +45.103, E3 +350633.871}
SPL {X  -165.650, Y  +415.564, Z    +0.000, E1   +45.195, E3 +350647.410}
SPL {X  -165.650, Y  +410.687, Z    +0.000, E1   +44.955, E3 +350658.726}
SPL {X  -165.650, Y  +405.522, Z    +0.000, E1   +45.119, E3 +350668.287}
SPL {X  -165.650, Y  +399.216, Z    +0.000, E1   +45.246, E3 +350680.480}
SPL {X  -165.650, Y  +391.618, Z    +0.000, E1   +45.037, E3 +350697.259}
SPL {X  -165.650, Y  +383.700, Z    +0.000, E1   +45.345, E3 +350711.385}
SPL {X  -165.650, Y  +379.225, Z    +0.000, E1   +45.073, E3 +350722.074}
SPL {X  -165.591, Y  +374.097, Z    +0.000, E1   +45.069, E3 +350732.555}
SPL {X  -165.372, Y  +368.914, Z    +0.000, E1   +45.103, E3 +350742.915}
SPL {X  -164.987, Y  +363.696, Z    +0.000, E1   +45.006, E3 +350754.138}
SPL {X  -164.256, Y  +357.053, Z    +0.000, E1   +44.969, E3 +350767.941}
SPL {X  -163.441, Y  +351.538, Z    +0.000, E1   +44.749, E3 +350780.304}
SPL {X  -162.419, Y  +345.942, Z    +0.000, E1   +44.540, E3 +350793.036}
SPL {X  -161.210, Y  +340.404, Z    +0.000, E1   +44.250, E3 +350805.861}
SPL {X  -159.961, Y  +335.460, Z    +0.000, E1   +44.205, E3 +350816.224}
SPL {X  -158.595, Y  +330.672, Z    +0.000, E1   +43.797, E3 +350828.202}
SPL {X  -156.695, Y  +324.773, Z    +0.000, E1   +43.987, E3 +350839.099}
SPL {X  -148.318, Y  +304.733, Z    +0.000, E1   +49.897, E3 +350844.336}
SPL {X  -138.435, Y  +287.529, Z    +0.000, E1   +45.834, E3 +350909.660}
SPL {X  -134.645, Y  +282.008, Z    +0.000, E1   +45.207, E3 +350939.316}
ENDSPLINE

SPLINE
SPL {X  -154.915, Y  +319.839, Z    +0.000, E1   +31.584, E3 +350998.836}
SPL {X  -161.387, Y  +341.161, Z    +0.000, E1   +22.590, E3 +351012.681}
SPL {X  -164.566, Y  +359.576, Z    +0.000, E1   +13.425, E3 +350991.274}
SPL {X  -165.355, Y  +368.611, Z    +0.000, E1    +8.407, E3 +350994.855}
SPL {X  -165.614, Y  +375.050, Z    +0.000, E1    +4.520, E3 +350996.159}
SPL {X  -165.650, Y  +379.271, Z    +0.000, E1    +1.752, E3 +350993.181}
SPL {X  -165.650, Y  +382.603, Z    +0.000, E1    -0.657, E3 +350994.389}
SPL {X  -165.650, Y  +386.866, Z    +0.000, E1    -4.337, E3 +350993.654}
SPL {X  -165.650, Y  +394.200, Z    +0.000, E1   -11.943, E3 +350991.421}
SPL {X  -165.650, Y  +405.401, Z    +0.000, E1   -24.512, E3 +350991.242}
SPL {X  -165.650, Y  +418.038, Z    +0.000, E1   -38.688, E3 +350987.469}
SPL {X  -165.650, Y  +461.620, Z    +0.000, E1   -55.594, E3 +351007.648}
SPL {X  -165.650, Y  +498.574, Z    +0.000, E1   -52.082, E3 +351068.673}
ENDSPLINE

SPLINE
SPL {X  -165.650, Y  +483.168, Z    +0.000, E1   -45.573, E3 +351079.330}
ENDSPLINE

SPLINE
SPL {X  -165.650, Y  +487.615, Z    +0.000, E1   -45.254, E3 +351090.351}
SPL {X  -165.650, Y  +493.602, Z    +0.000, E1   -45.283, E3 +351102.191}
SPL {X  -165.650, Y  +498.857, Z    +0.000, E1   -45.339, E3 +351112.535}
SPL {X  -165.650, Y  +504.159, Z    +0.000, E1   -45.384, E3 +351122.930}
SPL {X  -165.650, Y  +509.628, Z    +0.000, E1   -45.217, E3 +351135.113}
SPL {X  -165.650, Y  +516.157, Z    +0.000, E1   -45.240, E3 +351148.148}
SPL {X  -165.650, Y  +521.049, Z    +0.000, E1   -45.236, E3 +351158.101}
SPL {X  -165.650, Y  +527.050, Z    +0.000, E1   -45.345, E3 +351169.597}
SPL {X  -165.650, Y  +532.042, Z    +0.000, E1   -45.233, E3 +351180.341}
SPL {X  -165.650, Y  +537.290, Z    +0.000, E1   -45.204, E3 +351191.182}
SPL {X  -165.650, Y  +544.196, Z    +0.000, E1   -45.432, E3 +351203.856}
SPL {X  -165.650, Y  +548.678, Z    +0.000, E1   -45.162, E3 +351214.420}
SPL {X  -165.650, Y  +554.600, Z    +0.000, E1   -45.345, E3 +351225.397}
SPL {X  -165.650, Y  +559.896, Z    +0.000, E1   -45.150, E3 +351237.252}
SPL {X  -165.650, Y  +566.830, Z    +0.000, E1   -45.346, E3 +351250.232}
SPL {X  -165.650, Y  +575.003, Z    +0.000, E1   -45.370, E3 +351266.717}
SPL {X  -165.650, Y  +583.131, Z    +0.000, E1   -45.255, E3 +351283.768}
SPL {X  -165.650, Y  +590.060, Z    +0.000, E1   -45.221, E3 +351297.962}
SPL {X  -165.650, Y  +596.611, Z    +0.000, E1   -45.390, E3 +351310.199}
SPL {X  -165.650, Y  +601.960, Z    +0.000, E1   -45.255, E3 +351321.807}
SPL {X  -165.650, Y  +605.976, Z    +0.000, E1   -45.260, E3 +351329.857}
SPL {X  -165.650, Y  +610.850, Z    +0.000, E1   -45.208, E3 +351340.125}
SPL {X  -165.650, Y  +617.450, Z    +0.000, E1   -45.402, E3 +351352.328}
SPL {X  -165.650, Y  +622.720, Z    +0.000, E1   -45.272, E3 +351363.726}
SPL {X  -165.650, Y  +627.828, Z    +0.000, E1   -45.174, E3 +351374.682}
SPL {X  -165.650, Y  +634.620, Z    +0.000, E1   -45.438, E3 +351386.888}
SPL {X  -165.650, Y  +640.808, Z    +0.000, E1   -45.294, E3 +351400.262}
SPL {X  -165.650, Y  +646.552, Z    +0.000, E1   -45.137, E3 +351412.787}
SPL {X  -165.650, Y  +652.431, Z    +0.000, E1   -45.333, E3 +351423.541}
SPL {X  -165.650, Y  +657.443, Z    +0.000, E1   -45.316, E3 +351433.797}
SPL {X  -165.650, Y  +662.999, Z    +0.000, E1   -45.214, E3 +351445.669}
SPL {X  -165.650, Y  +668.737, Z    +0.000, E1   -45.236, E3 +351457.184}
SPL {X  -165.650, Y  +675.226, Z    +0.000, E1   -45.503, E3 +351468.688}
SPL {X  -165.597, Y  +679.672, Z    +0.000, E1   -45.206, E3 +351479.409}
SPL {X  -165.388, Y  +684.808, Z    +0.000, E1   -45.192, E3 +351489.917}
SPL {X  -165.020, Y  +689.938, Z    +0.000, E1   -45.107, E3 +351500.859}
SPL {X  -164.358, Y  +696.147, Z    +0.000, E1   -45.160, E3 +351513.125}
SPL {X  -163.631, Y  +701.286, Z    +0.000, E1   -44.994, E3 +351524.417}
SPL {X  -163.047, Y  +704.748, Z    +0.000, E1   -44.682, E3 +351533.241}
SPL {X  -161.884, Y  +710.619, Z    +0.000, E1   -44.738, E3 +351544.866}
SPL {X  -160.692, Y  +715.726, Z    +0.000, E1   -44.379, E3 +351557.188}
SPL {X  -158.938, Y  +722.175, Z    +0.000, E1   -44.121, E3 +351571.836}
SPL {X  -156.604, Y  +729.490, Z    +0.000, E1   -44.229, E3 +351585.826}
SPL {X  -147.100, Y  +751.668, Z    +0.000, E1   -50.624, E3 +351591.713}
SPL {X  -144.116, Y  +757.172, Z    +0.000, E1   -42.809, E3 +351661.109}
SPL {X  -127.227, Y  +781.582, Z    +0.000, E1   -46.780, E3 +351706.779}
ENDSPLINE

SPLINE
SPL {X  -133.736, Y  +773.248, Z    +0.000, E1   -45.385, E3 +351784.821}
SPL {X  -160.761, Y  +715.447, Z    +0.000, E1   -23.748, E3 +351741.671}
SPL {X  -164.304, Y  +696.571, Z    +0.000, E1   -14.525, E3 +351746.895}
SPL {X  -165.498, Y  +682.585, Z    +0.000, E1    -6.769, E3 +351746.569}
SPL {X  -165.650, Y  +674.975, Z    +0.000, E1    -1.888, E3 +351744.928}
SPL {X  -165.650, Y  +671.520, Z    +0.000, E1    +0.682, E3 +351743.855}
SPL {X  -165.650, Y  +668.289, Z    +0.000, E1    +3.417, E3 +351743.697}
SPL {X  -165.650, Y  +663.040, Z    +0.000, E1    +8.602, E3 +351742.891}
SPL {X  -165.650, Y  +655.692, Z    +0.000, E1   +17.061, E3 +351741.427}
SPL {X  -165.650, Y  +646.511, Z    +0.000, E1   +26.434, E3 +351744.207}
SPL {X  -165.650, Y  +637.905, Z    +0.000, E1   +40.225, E3 +351732.331}
SPL {X  -165.650, Y  +607.385, Z    +0.000, E1   +51.775, E3 +351752.089}
SPL {X  -165.650, Y  +598.058, Z    +0.000, E1   +51.157, E3 +351765.551}
SPL {X  -165.650, Y  +553.219, Z    +0.000, E1   +52.865, E3 +351819.733}
ENDSPLINE

SPLINE
SPL {X  -165.650, Y  +569.883, Z    +0.000, E1   +45.183, E3 +351835.410}
ENDSPLINE

SPLINE
SPL {X  -165.650, Y  +564.081, Z    +0.000, E1   +45.208, E3 +351847.028}
SPL {X  -165.650, Y  +559.277, Z    +0.000, E1   +45.277, E3 +351856.319}
SPL {X  -165.650, Y  +554.065, Z    +0.000, E1   +45.254, E3 +351867.128}
SPL {X  -165.650, Y  +548.074, Z    +0.000, E1   +45.245, E3 +351879.238}
SPL {X  -165.650, Y  +542.958, Z    +0.000, E1   +45.131, E3 +351890.369}
SPL {X  -165.650, Y  +535.288, Z    +0.000, E1   +45.332, E3 +351904.810}
SPL {X  -165.650, Y  +528.026, Z    +0.000, E1   +45.173, E3 +351920.468}
SPL {X  -165.650, Y  +520.964, Z    +0.000, E1   +45.458, E3 +351932.974}
SPL {X  -165.650, Y  +516.211, Z    +0.000, E1   +45.175, E3 +351944.316}
SPL {X  -165.650, Y  +509.762, Z    +0.000, E1   +45.191, E3 +351957.359}
SPL {X  -165.650, Y  +503.812, Z    +0.000, E1   +45.188, E3 +351969.397}
SPL {X  -165.650, Y  +499.646, Z    +0.000, E1   +44.886, E3 +351979.668}
ENDSPLINE

SPLINE
SPL {X  -165.650, Y  +516.930, Z    +0.000, E1   +36.544, E3 +351988.339}
ENDSPLINE

SPLINE
SPL {X  -165.650, Y  +511.324, Z    +0.000, E1   +37.254, E3 +351999.330}
SPL {X  -165.650, Y  +502.734, Z    +0.000, E1   +38.389, E3 +352015.098}
SPL {X  -165.650, Y  +493.826, Z    +0.000, E1   +39.521, E3 +352030.761}
SPL {X  -165.650, Y  +487.003, Z    +0.000, E1   +40.380, E3 +352042.216}
SPL {X  -165.650, Y  +478.382, Z    +0.000, E1   +41.628, E3 +352055.128}
SPL {X  -165.650, Y  +468.596, Z    +0.000, E1   +42.673, E3 +352071.035}
SPL {X  -165.650, Y  +458.202, Z    +0.000, E1   +44.020, E3 +352085.576}
SPL {X  -165.650, Y  +449.099, Z    +0.000, E1   +44.871, E3 +352099.538}
SPL {X  -165.650, Y  +442.120, Z    +0.000, E1   +45.313, E3 +352111.090}
SPL {X  -165.650, Y  +439.103, Z    +0.000, E1   +44.726, E3 +352120.699}
SPL {X  -165.650, Y  +433.421, Z    +0.000, E1   +45.110, E3 +352130.086}
SPL {X  -165.650, Y  +427.943, Z    +0.000, E1   +45.362, E3 +352139.711}
SPL {X  -165.650, Y  +422.523, Z    +0.000, E1   +45.103, E3 +352152.390}
SPL {X  -165.650, Y  +415.564, Z    +0.000, E1   +45.195, E3 +352165.929}
SPL {X  -165.650, Y  +410.687, Z    +0.000, E1   +44.955, E3 +352177.245}
SPL {X  -165.650, Y  +402.778, Z    +0.000, E1   +45.323, E3 +352191.326}
SPL {X  -165.650, Y  +396.171, Z    +0.000, E1   +44.969, E3 +352206.746}
SPL {X  -165.650, Y  +390.060, Z    +0.000, E1   +45.007, E3 +352218.980}
SPL {X  -165.650, Y  +383.700, Z    +0.000, E1   +45.345, E3 +352229.904}
SPL {X  -165.650, Y  +379.225, Z    +0.000, E1   +45.073, E3 +352240.593}
SPL {X  -165.591, Y  +374.097, Z    +0.000, E1   +45.069, E3 +352251.074}
SPL {X  -165.372, Y  +368.914, Z    +0.000, E1   +45.103, E3 +352261.434}
SPL {X  -164.833, Y  +362.064, Z    +0.000, E1   +44.999, E3 +352276.219}
SPL {X  -164.024, Y  +355.348, Z    +0.000, E1   +45.002, E3 +352289.607}
SPL {X  -163.441, Y  +351.538, Z    +0.000, E1   +44.749, E3 +352298.823}
SPL {X  -162.419, Y  +345.942, Z    +0.000, E1   +44.540, E3 +352311.555}
SPL {X  -161.210, Y  +340.404, Z    +0.000, E1   +44.250, E3 +352324.379}
SPL {X  -159.961, Y  +335.460, Z    +0.000, E1   +44.205, E3 +352334.742}
SPL {X  -158.595, Y  +330.672, Z    +0.000, E1   +43.797, E3 +352346.721}
SPL {X  -157.207, Y  +326.289, Z    +0.000, E1   +43.631, E3 +352356.474}
SPL {X  -152.192, Y  +313.097, Z    +0.000, E1   +47.715, E3 +352360.027}
SPL {X  -146.385, Y  +300.967, Z    +0.000, E1   +50.402, E3 +352366.223}
SPL {X  -138.435, Y  +287.529, Z    +0.000, E1   +45.834, E3 +352428.179}
SPL {X  -134.645, Y  +282.008, Z    +0.000, E1   +45.207, E3 +352457.835}
ENDSPLINE

SPLINE
SPL {X  -154.915, Y  +319.839, Z    +0.000, E1   +31.584, E3 +352517.354}
SPL {X  -161.387, Y  +341.161, Z    +0.000, E1   +22.590, E3 +352531.199}
SPL {X  -164.566, Y  +359.576, Z    +0.000, E1   +13.425, E3 +352509.793}
SPL {X  -165.355, Y  +368.611, Z    +0.000, E1    +8.407, E3 +352513.374}
SPL {X  -165.614, Y  +375.050, Z    +0.000, E1    +4.520, E3 +352514.677}
SPL {X  -165.650, Y  +379.847, Z    +0.000, E1    +1.364, E3 +352513.027}
SPL {X  -165.650, Y  +383.246, Z    +0.000, E1    -1.216, E3 +352512.120}
SPL {X  -165.650, Y  +386.866, Z    +0.000, E1    -4.337, E3 +352512.173}
SPL {X  -165.650, Y  +394.200, Z    +0.000, E1   -11.943, E3 +352509.940}
SPL {X  -165.650, Y  +405.401, Z    +0.000, E1   -24.512, E3 +352509.760}
SPL {X  -165.650, Y  +418.038, Z    +0.000, E1   -38.688, E3 +352505.987}
SPL {X  -165.650, Y  +461.620, Z    +0.000, E1   -55.594, E3 +352526.166}
SPL {X  -165.650, Y  +498.574, Z    +0.000, E1   -52.082, E3 +352587.191}
ENDSPLINE

SPLINE
SPL {X  -165.650, Y  +484.983, Z    +0.000, E1   -45.406, E3 +352602.694}
ENDSPLINE

SPLINE
SPL {X  -165.650, Y  +492.090, Z    +0.000, E1   -45.292, E3 +352617.717}
SPL {X  -165.650, Y  +498.857, Z    +0.000, E1   -45.339, E3 +352631.054}
SPL {X  -165.650, Y  +505.115, Z    +0.000, E1   -45.299, E3 +352644.002}
SPL {X  -165.650, Y  +510.931, Z    +0.000, E1   -45.250, E3 +352655.993}
SPL {X  -165.650, Y  +516.157, Z    +0.000, E1   -45.240, E3 +352666.667}
SPL {X  -165.650, Y  +521.049, Z    +0.000, E1   -45.236, E3 +352676.620}
SPL {X  -165.650, Y  +527.050, Z    +0.000, E1   -45.345, E3 +352688.116}
SPL {X  -165.650, Y  +532.042, Z    +0.000, E1   -45.233, E3 +352698.859}
SPL {X  -165.650, Y  +537.290, Z    +0.000, E1   -45.204, E3 +352709.700}
SPL {X  -165.650, Y  +544.196, Z    +0.000, E1   -45.432, E3 +352722.374}
SPL {X  -165.650, Y  +548.678, Z    +0.000, E1   -45.162, E3 +352732.938}
SPL {X  -165.650, Y  +554.600, Z    +0.000, E1   -45.345, E3 +352743.915}
SPL {X  -165.650, Y  +559.896, Z    +0.000, E1   -45.150, E3 +352755.770}
SPL {X  -165.650, Y  +566.830, Z    +0.000, E1   -45.346, E3 +352768.751}
SPL {X  -165.650, Y  +573.074, Z    +0.000, E1   -45.379, E3 +352781.081}
SPL {X  -165.650, Y  +579.360, Z    +0.000, E1   -45.300, E3 +352794.367}
SPL {X  -165.650, Y  +584.577, Z    +0.000, E1   -45.167, E3 +352805.590}
SPL {X  -165.650, Y  +590.060, Z    +0.000, E1   -45.221, E3 +352816.481}
SPL {X  -165.650, Y  +596.611, Z    +0.000, E1   -45.390, E3 +352828.717}
SPL {X  -165.650, Y  +603.637, Z    +0.000, E1   -45.296, E3 +352843.636}
SPL {X  -165.650, Y  +610.850, Z    +0.000, E1   -45.208, E3 +352858.644}
SPL {X  -165.650, Y  +617.450, Z    +0.000, E1   -45.402, E3 +352870.846}
SPL {X  -165.650, Y  +622.720, Z    +0.000, E1   -45.272, E3 +352882.244}
SPL {X  -165.650, Y  +627.828, Z    +0.000, E1   -45.174, E3 +352893.201}
SPL {X  -165.650, Y  +634.620, Z    +0.000, E1   -45.438, E3 +352905.406}
SPL {X  -165.650, Y  +640.808, Z    +0.000, E1   -45.294, E3 +352918.781}
SPL {X  -165.650, Y  +646.552, Z    +0.000, E1   -45.137, E3 +352931.305}
SPL {X  -165.650, Y  +652.431, Z    +0.000, E1   -45.333, E3 +352942.060}
SPL {X  -165.650, Y  +657.443, Z    +0.000, E1   -45.316, E3 +352952.316}
SPL {X  -165.650, Y  +662.999, Z    +0.000, E1   -45.214, E3 +352964.188}
SPL {X  -165.650, Y  +668.737, Z    +0.000, E1   -45.236, E3 +352975.703}
SPL {X  -165.650, Y  +675.226, Z    +0.000, E1   -45.503, E3 +352987.206}
SPL {X  -165.597, Y  +679.672, Z    +0.000, E1   -45.206, E3 +352997.928}
SPL {X  -165.388, Y  +684.808, Z    +0.000, E1   -45.192, E3 +353008.435}
SPL {X  -165.020, Y  +689.938, Z    +0.000, E1   -45.107, E3 +353019.378}
SPL {X  -164.358, Y  +696.147, Z    +0.000, E1   -45.160, E3 +353031.644}
SPL {X  -163.631, Y  +701.286, Z    +0.000, E1   -44.994, E3 +353042.936}
SPL {X  -162.679, Y  +706.734, Z    +0.000, E1   -44.812, E3 +353055.169}
SPL {X  -161.655, Y  +711.661, Z    +0.000, E1   -44.525, E3 +353066.550}
SPL {X  -160.692, Y  +715.726, Z    +0.000, E1   -44.379, E3 +353075.707}
SPL {X  -159.384, Y  +720.631, Z    +0.000, E1   -44.155, E3 +353086.857}
SPL {X  -158.321, Y  +724.227, Z    +0.000, E1   -43.955, E3 +353095.178}
SPL {X  -156.604, Y  +729.490, Z    +0.000, E1   -44.229, E3 +353104.345}
SPL {X  -147.100, Y  +751.668, Z    +0.000, E1   -50.624, E3 +353110.232}
SPL {X  -144.116, Y  +757.172, Z    +0.000, E1   -42.809, E3 +353179.628}
SPL {X  -127.227, Y  +781.582, Z    +0.000, E1   -46.780, E3 +353225.297}
ENDSPLINE

